// TwinCAT 3 PLC project FRA3
// libraries:
//   Tc2_DataExchange, * (Beckhoff Automation GmbH)
//   Tc2_Standard, * (Beckhoff Automation GmbH)
//   Tc2_System, * (Beckhoff Automation GmbH)
//   Tc2_Utilities, * (Beckhoff Automation GmbH)
//   Tc3_Module, * (Beckhoff Automation GmbH)
//   VisuSymbols,3.5.10.0,System
// project tree:
//   Global Variables/ Global_Variables.TcGVL, Global_Variables_HMI.TcGVL, GVAR_Control.TcGVL, GVAR_Status_and_Alarms.TcGVL, Variable_Configuration.TcGVL
//   POUs/ Control.TcPOU, Hopper_Level.TcPOU, MAIN.TcPOU, Messages.TcPOU, Production_Runtime_Values.TcPOU, Runtime_Control.TcPOU, Speed_Setpoints.TcPOU, StandardCPM.TcPOU, Status_and_Alarms.TcPOU
//   POUs/Function Blocks/ CheckDiv_1.TcPOU, Codes_StopReason.TcPOU, CounterEx.TcPOU, FB_Downtime_LOG.TcPOU, FillerCPM_Current.TcPOU, FixedSchedule_FillerRoom.TcPOU, GetTime_Seconds.TcPOU, LimitRealNumber.TcPOU, LimitRealNumberToWord.TcPOU, ScaleWithParameters.TcPOU, StandardCPMSet.TcPOU, TOGGLE.TcPOU
//   / Standard.TcTTO
// real-time tasks:
//   TASK Standard: cycle T#10ms, priority 20, ADS port 350
// I/O:
//   DEVICE FRA 3 I/O, AmsNetId 5.176.210.24.2.1
//     Term 1 (EK1200) [EK1200-7000 EtherCAT Power supply (1,5A E-Bus)]
//       Term 2 (EL1018) [EL1018 8Ch. Dig. Input 24V, 10µs]
//       Term 3 (EL1018) [EL1018 8Ch. Dig. Input 24V, 10µs]
//       Term 4 (EL1018) [EL1018 8Ch. Dig. Input 24V, 10µs]
//       Term 5 (EL4022) [EL4022 2Ch. Ana. Output 4-20mA, 12bit]
//       Term 6 (EL4022) [EL4022 2Ch. Ana. Output 4-20mA, 12bit]
//       Term 7 (EL4022) [EL4022 2Ch. Ana. Output 4-20mA, 12bit]
//       Term 8 (EL4022) [EL4022 2Ch. Ana. Output 4-20mA, 12bit]
//       Term 9 (EL4022) [EL4022 2Ch. Ana. Output 4-20mA, 12bit]
//       Term 10 (EL4022) [EL4022 2Ch. Ana. Output 4-20mA, 12bit]
//       Term 11 (EL3052) [EL3052 2Ch. Ana. Input 4-20mA]
//       Term 12 (EL3202) [EL3202 2Ch. Ana. Input PT100 (RTD)]
//       Term 13 (EL9110) [EL9110 Power Supplier with LED (24V, Diagnostics)]
//       Term 14 (EL9160) [EL9160 Power Supplier with LED (230V, Diagnostics)]
//       Term 15 (EL2602) [EL2602 2Ch. Relay Output, NO (230V AC / 30V DC)]
//       Term 16 (EL2602) [EL2602 2Ch. Relay Output, NO (230V AC / 30V DC)]
//       Term 17 (EL2602) [EL2602 2Ch. Relay Output, NO (230V AC / 30V DC)]
//       Term 18 (EL2612) [EL2612 2Ch. Relay Output, CO (125V AC / 30V DC)]
//       Term 19 (EL2612) [EL2612 2Ch. Relay Output, CO (125V AC / 30V DC)]
//       Term 20 (EL2612) [EL2612 2Ch. Relay Output, CO (125V AC / 30V DC)]
//       Term 21 (EL2612) [EL2612 2Ch. Relay Output, CO (125V AC / 30V DC)]
//       Term 22 (EL2612) [EL2612 2Ch. Relay Output, CO (125V AC / 30V DC)]
//       Term 23 (EL2612) [EL2612 2Ch. Relay Output, CO (125V AC / 30V DC)]
//       Term 24 (EL2612) [EL2612 2Ch. Relay Output, CO (125V AC / 30V DC)]
//       Term 25 (EL2612) [EL2612 2Ch. Relay Output, CO (125V AC / 30V DC)]
//       Term 26 (EL2612) [EL2612 2Ch. Relay Output, CO (125V AC / 30V DC)]
//       Term 27 (EL9011) [EL9011 End Terminal]
// variable links:
//   FRA3/FRA3 Instance <-> FRA 3 I/O/Term 1 (EK1200)/Term 10 (EL4022)
//     Standard Outputs/.oBrine_Tank_Steam <-> AO Outputs Channel 2/.oBrine_Tank_Steam
//     Standard Outputs/.oSpiral_Infeed_Spd <-> AO Outputs Channel 1/.oSpiral_Infeed_Spd
//   FRA3/FRA3 Instance <-> FRA 3 I/O/Term 1 (EK1200)/Term 11 (EL3052)
//     Standard Inputs/.iHopper_Level <-> AI Standard Channel 1/.iHopper_Level
//   FRA3/FRA3 Instance <-> FRA 3 I/O/Term 1 (EK1200)/Term 12 (EL3202)
//     Standard Inputs/.i1062 <-> RTD Inputs Channel 2/.i1062
//     Standard Inputs/.iSpice_Tank_Temp <-> RTD Inputs Channel 1/.iSpice_Tank_Temp
//   FRA3/FRA3 Instance <-> FRA 3 I/O/Term 1 (EK1200)/Term 14 (EL9160)
//     Standard Inputs/.iEmergency_Stop <-> PowerOK/.iEmergency_Stop
//   FRA3/FRA3 Instance <-> FRA 3 I/O/Term 1 (EK1200)/Term 15 (EL2602)
//     Standard Outputs/.oPreBrine_Flap <-> Channel 2/.oPreBrine_Flap
//     Standard Outputs/.oReturn_Pump <-> Channel 1/.oReturn_Pump
//   FRA3/FRA3 Instance <-> FRA 3 I/O/Term 1 (EK1200)/Term 16 (EL2602)
//     Standard Outputs/.oPre_Brine <-> Channel 1/.oPre_Brine
//     Standard Outputs/.oWater_Valve <-> Channel 2/.oWater_Valve
//   FRA3/FRA3 Instance <-> FRA 3 I/O/Term 1 (EK1200)/Term 17 (EL2602)
//     Standard Outputs/.oBrine_Flap <-> Channel 2/.oBrine_Flap
//     Standard Outputs/.oCloser_Clutch_Sol <-> Channel 1/.oCloser_Clutch_Sol
//   FRA3/FRA3 Instance <-> FRA 3 I/O/Term 1 (EK1200)/Term 18 (EL2612)
//     Standard Outputs/.o1801 <-> Channel 2/.o1801
//     Standard Outputs/.oSpiral_Infeed <-> Channel 1/.oSpiral_Infeed
//   FRA3/FRA3 Instance <-> FRA 3 I/O/Term 1 (EK1200)/Term 19 (EL2612)
//     Standard Outputs/.oCloser <-> Channel 2/.oCloser
//     Standard Outputs/.oSpiral <-> Channel 1/.oSpiral
//   FRA3/FRA3 Instance <-> FRA 3 I/O/Term 1 (EK1200)/Term 2 (EL1018)
//     Standard Inputs/.F_Closer <-> Channel 2/.F_Closer
//     Standard Inputs/.F_Elevator <-> Channel 1/.F_Elevator
//     Standard Inputs/.F_Empty_Can_Conv <-> Channel 8/.F_Empty_Can_Conv
//     Standard Inputs/.F_Empty_Can_Track <-> Channel 7/.F_Empty_Can_Track
//     Standard Inputs/.F_Engler_Filler <-> Channel 5/.F_Engler_Filler
//     Standard Inputs/.F_Full_Can_Belt <-> Channel 3/.F_Full_Can_Belt
//     Standard Inputs/.F_Juicer <-> Channel 4/.F_Juicer
//     Standard Inputs/.F_Twin_Auger <-> Channel 6/.F_Twin_Auger
//   FRA3/FRA3 Instance <-> FRA 3 I/O/Term 1 (EK1200)/Term 20 (EL2612)
//     Standard Outputs/.oFull_Can_Belt <-> Channel 1/.oFull_Can_Belt
//     Standard Outputs/.oJuicer <-> Channel 2/.oJuicer
//   FRA3/FRA3 Instance <-> FRA 3 I/O/Term 1 (EK1200)/Term 21 (EL2612)
//     Standard Outputs/.oEngler_Filler <-> Channel 1/.oEngler_Filler
//     Standard Outputs/.oTwin_Auger_Forward <-> Channel 2/.oTwin_Auger_Forward
//   FRA3/FRA3 Instance <-> FRA 3 I/O/Term 1 (EK1200)/Term 22 (EL2612)
//     Standard Outputs/.oOutfeed_Can_Belt <-> Channel 2/.oOutfeed_Can_Belt
//     Standard Outputs/.oTwin_Auger_Reverse <-> Channel 1/.oTwin_Auger_Reverse
//   FRA3/FRA3 Instance <-> FRA 3 I/O/Term 1 (EK1200)/Term 23 (EL2612)
//     Standard Outputs/.oEmpty_Can_Conv <-> Channel 2/.oEmpty_Can_Conv
//     Standard Outputs/.oEmpty_Can_Track <-> Channel 1/.oEmpty_Can_Track
//   FRA3/FRA3 Instance <-> FRA 3 I/O/Term 1 (EK1200)/Term 24 (EL2612)
//     Standard Outputs/.oInfeed_Auger_Fwd <-> Channel 1/.oInfeed_Auger_Fwd
//     Standard Outputs/.oInfeed_Auger_Rev <-> Channel 2/.oInfeed_Auger_Rev
//   FRA3/FRA3 Instance <-> FRA 3 I/O/Term 1 (EK1200)/Term 25 (EL2612)
//     Standard Outputs/.oCloser_ButtonLt <-> Channel 2/.oCloser_ButtonLt
//     Standard Outputs/.oStatusLt <-> Channel 1/.oStatusLt
//   FRA3/FRA3 Instance <-> FRA 3 I/O/Term 1 (EK1200)/Term 26 (EL2612)
//     Standard Outputs/.oPreBrine_Overflow_Pump <-> Channel 2/.oPreBrine_Overflow_Pump
//     Standard Outputs/.oSpiral_ButtonLt <-> Channel 1/.oSpiral_ButtonLt
//   FRA3/FRA3 Instance <-> FRA 3 I/O/Term 1 (EK1200)/Term 3 (EL1018)
//     Standard Inputs/.F_Exit_Conveyor <-> Channel 6/.F_Exit_Conveyor
//     Standard Inputs/.F_Infeed_Auger <-> Channel 7/.F_Infeed_Auger
//     Standard Inputs/.i403 <-> Channel 8/.i403
//     Standard Inputs/.iCloser_Can_Jam <-> Channel 5/.iCloser_Can_Jam
//     Standard Inputs/.iCloser_Start_PB <-> Channel 2/.iCloser_Start_PB
//     Standard Inputs/.iElevator_Start_PB <-> Channel 3/.iElevator_Start_PB
//     Standard Inputs/.iEmpty_Can_Sensor <-> Channel 4/.iEmpty_Can_Sensor
//     Standard Inputs/.iSpice_Tank_Level <-> Channel 1/.iSpice_Tank_Level
//   FRA3/FRA3 Instance <-> FRA 3 I/O/Term 1 (EK1200)/Term 4 (EL1018)
//     Standard Inputs/.i601 <-> Channel 6/.i601
//     Standard Inputs/.i602 <-> Channel 7/.i602
//     Standard Inputs/.iCloser_Speed_Pulse <-> Channel 8/.iCloser_Speed_Pulse
//     Standard Inputs/.iDischarge_Can_Jam <-> Channel 2/.iDischarge_Can_Jam
//     Standard Inputs/.iElevator_Jam_Sensor <-> Channel 1/.iElevator_Jam_Sensor
//     Standard Inputs/.iPreBrine_Tank_Level <-> Channel 3/.iPreBrine_Tank_Level
//     Standard Inputs/.iSpiral_Can_Counter <-> Channel 5/.iSpiral_Can_Counter
//     Standard Inputs/.iSteamPressSwitch <-> Channel 4/.iSteamPressSwitch
//   FRA3/FRA3 Instance <-> FRA 3 I/O/Term 1 (EK1200)/Term 5 (EL4022)
//     Standard Outputs/.oCloser_Speed <-> AO Outputs Channel 2/.oCloser_Speed
//     Standard Outputs/.oSpice_Pump_Speed <-> AO Outputs Channel 1/.oSpice_Pump_Speed
//   FRA3/FRA3 Instance <-> FRA 3 I/O/Term 1 (EK1200)/Term 6 (EL4022)
//     Standard Outputs/.oElevator_Speed <-> AO Outputs Channel 1/.oElevator_Speed
//     Standard Outputs/.oFull_Can_Belt_Speed <-> AO Outputs Channel 2/.oFull_Can_Belt_Speed
//   FRA3/FRA3 Instance <-> FRA 3 I/O/Term 1 (EK1200)/Term 7 (EL4022)
//     Standard Outputs/.oEngler_Filler_Speed <-> AO Outputs Channel 1/.oEngler_Filler_Speed
//     Standard Outputs/.oTwin_Auger_Speed <-> AO Outputs Channel 2/.oTwin_Auger_Speed
//   FRA3/FRA3 Instance <-> FRA 3 I/O/Term 1 (EK1200)/Term 8 (EL4022)
//     Standard Outputs/.oEmpty_Can_Track_Spd <-> AO Outputs Channel 2/.oEmpty_Can_Track_Spd
//     Standard Outputs/.oExit_Conv_Speed <-> AO Outputs Channel 1/.oExit_Conv_Speed
//   FRA3/FRA3 Instance <-> FRA 3 I/O/Term 1 (EK1200)/Term 9 (EL4022)
//     Standard Outputs/.oEmpty_Can_Conv_Spd <-> AO Outputs Channel 1/.oEmpty_Can_Conv_Spd
//     Standard Outputs/.oInfeed_Auger <-> AO Outputs Channel 2/.oInfeed_Auger

CONFIGURATION FRA3
    RESOURCE PLC ON TwinCAT3
        TASK Standard(INTERVAL := T#10ms, PRIORITY := 20);
        PROGRAM MAIN WITH Standard : MAIN;
    END_RESOURCE
END_CONFIGURATION

// ---- Global Variables/Global_Variables.TcGVL
{attribute 'Tc2GvlVarNames'}
VAR_GLOBAL 
(*****Fill Room A-2****)

(****Slot 1 KL-3052****)
	iHopper_Level AT %I* : WORD;
	i004 AT %I* : WORD;

(****Slot 2 KL-1114****)
	F_Elevator AT %I* : BOOL;
	F_Closer AT %I* : BOOL;
	F_Full_Can_Belt AT %I* : BOOL;
	F_Juicer AT %I* : BOOL;

(****Slot 3 KL-1114****)
	F_Engler_Filler AT %I* : BOOL;
	F_Twin_Auger AT %I* : BOOL;
	F_Empty_Can_Track AT %I* : BOOL;
	F_Empty_Can_Conv AT %I* : BOOL;

(****Slot 4 KL-1114****)
	iSpice_Tank_Level AT %I* : BOOL;
	iCloser_Start_PB AT %I* : BOOL;
	iElevator_Start_PB AT %I* : BOOL;
	iEmpty_Can_Sensor AT %I* : BOOL;

(****Slot 5 KL-1114****)
	iCloser_Can_Jam AT %I* : BOOL;
	F_Exit_Conveyor AT %I* : BOOL;
	F_Infeed_Auger AT %I* : BOOL;
	i403 AT %I* : BOOL;

(****Slot 6 KL-1114****)
	iElevator_Jam_Sensor AT %I* : BOOL;
	iDischarge_Can_Jam AT %I* : BOOL;
	iPreBrine_Tank_Level AT %I* : BOOL;
	iSteamPressSwitch AT %I* : BOOL;

(****Slot 7 KL-1114****)
	iSpiral_Can_Counter AT %I* : BOOL;
	i601 AT %I* : BOOL;
	i602 AT %I* : BOOL;
	iCloser_Speed_Pulse AT %I* : BOOL;

(****Slot 8 KL-4022****)
	oSpice_Pump_Speed AT %Q* : WORD;
	oCloser_Speed AT %Q* : WORD;

(****Slot 9 KL-4022****)
	oElevator_Speed AT %Q* : WORD;
	oFull_Can_Belt_Speed AT %Q* : WORD;

(****Slot 10 KL-4022****)
	oEngler_Filler_Speed AT %Q* : WORD;
	oTwin_Auger_Speed AT %Q* : WORD;

(****Slot 11 KL-4022****)
	oExit_Conv_Speed AT %Q* : WORD;
	oEmpty_Can_Track_Spd AT %Q* : WORD;

(****Slot 12 KL-4022****)
	oEmpty_Can_Conv_Spd AT %Q* : WORD;
	oInfeed_Auger AT %Q* : WORD;

(****Slot 13 KL-4022****)
	oSpiral_Infeed_Spd AT %Q* : WORD;
	oBrine_Tank_Steam AT %Q* : WORD;
	
(****Slot 15 KL-3052****)
	iTwinAugerLVL AT %I* : WORD;
	iSpare AT %I* : WORD;
	
(****Slot 14 KL-3202****)
	iSpice_Tank_Temp AT %I* : WORD;
	i1062 AT %I* : WORD;



(****Slot 16 KL-9260****)
	iEmergency_Stop AT %I* : BOOL;
	iPower AT %I* : BOOL;

(****Slot 17 KL-2602****)
	oReturn_Pump AT %Q* : BOOL;
	oPreBrine_Flap AT %Q* : BOOL;

(****Slot 18 KL-2602****)
	oPre_Brine AT %Q* : BOOL;
	oWater_Valve AT %Q* : BOOL;

(****Slot 19 KL-2602****)
	oCloser_Clutch_Sol AT %Q* : BOOL;
	oBrine_Flap AT %Q* : BOOL;

(****Slot 20 KL-2612****)
	oSpiral_Infeed AT %Q* : BOOL;
	o1801 AT %Q* : BOOL;

(****Slot 21 KL-2612****)
	oSpiral AT %Q* : BOOL;
	oCloser AT %Q* : BOOL;

(****Slot 22 KL-2612****)
	oFull_Can_Belt AT %Q* : BOOL;
	oJuicer AT %Q* : BOOL;

(****Slot 23 KL-2612****)
	oEngler_Filler AT %Q* : BOOL;
	oTwin_Auger_Forward AT %Q* : BOOL;

(****Slot 24 KL-2612****)
	oTwin_Auger_Reverse AT %Q* : BOOL;
	oOutfeed_Can_Belt AT %Q* : BOOL;

(****Slot 25 KL-2612****)
	oEmpty_Can_Track AT %Q* : BOOL;
	oEmpty_Can_Conv AT %Q* : BOOL;

(****Slot 26 KL-2612****)
	oInfeed_Auger_Fwd AT %Q* : BOOL;
	oInfeed_Auger_Rev AT %Q* : BOOL;

(****Slot 27 KL-2612****)
	oStatusLt AT %Q* : BOOL;
	oCloser_ButtonLt AT %Q* : BOOL;

(****Slot 28 KL-2612****)
	oSpiral_ButtonLt AT %Q* : BOOL;
	oPreBrine_Overflow_Pump AT %Q* : BOOL;

	Low_Spice_Alarm: BOOL;
	Low_Spice_Disable: BOOL;
	CleanMode: BOOL;
	Hopper_Level_PCT: REAL;
	TYLER: BOOL;
	Hopper_Level_High: BOOL;
	Brine_Temp_High: BOOL;
	Brine_Temp_Low: BOOL;
	Brine_Temp_Out_Of_Range: BOOL;
	Closer_Steam_Low_Disable: BOOL;
	CanCounter3: CTU;
	CC3Multiplier: CTU;
	DowntimeTotal_Min: REAL;
	EndRuntime: BOOL;
	AutoTog: TOGGLE;
	FillerPauseTog: TOGGLE;
	FillerAugerPause: TOGGLE;
	Empty_Can_Tog: TOGGLE;
	CC3Reset: BOOL;
	CanCntReset: BOOL;
	Count3: WORD;
    Runtime_Stopped: BOOL;
	Count3Real: REAL;
	MultiReal: REAL;
	HighCount: REAL;
	ActualCount: REAL;
	Cases: REAL;
    MultiWord: WORD ;

END_VAR

// ---- Global Variables/Global_Variables_HMI.TcGVL
{attribute 'Tc2GvlVarNames'}
VAR_GLOBAL

	s3ProdStd:REAL;

(*Speed Set Points*)
	sSpice_Pump_Speed_SPt: REAL;
	sCloser_Speed_SPt: REAL;
	sElevator_Speed_SPt: REAL;
	sFull_Can_Belt_Speed_SPt: REAL;
	sEngler_Filler_Speed_SPt: REAL;
	sTwin_Auger_Speed_SPt: REAL;
	sExit_Conveyor_Speed_SPt: REAL;
	Empty_Can_Track_SPt: REAL;
	Empty_Can_Conv_SPt: REAL;
	sInfeed_Auger_SPt: REAL;

(****Screen Activation****)

	sAuto: BOOL;
	sAuto_Run:BOOL;
	sAuto_Button : BOOL;
	sFiller_Pause_Button : BOOL;
	sFiller_Pause : BOOL;
	sFeed_Auger_Pause_Button : BOOL;
	sFeed_Auger_Pause : BOOL;
	sEmpty_Can_Track : BOOL;

	sFeed_Auger_Fwd : BOOL;
	sFeed_Auger_Rev : BOOL;
	sTwin_Auger_Fwd : BOOL;
	sTwin_Auger_Rev : BOOL;

	oInfeed_Auger_Fwd_Light: BOOL;
	oInfeed_Auger_Rev_Light: BOOL;
	oTwin_Auger_Forward_Light: BOOL;
	oTwin_Auger_Reverse_Light: BOOL;
	Jam_Fault: BOOL;
	sEngler_Filler : BOOL;
	sPreBrine : BOOL;
	sSpice_Tank_Fill : BOOL;
	sConveyors : BOOL;
	sJuicer : BOOL;
	sDiverter : BOOL;
	sEmpty_Can_Track_300A: BOOL;
	sCloser: BOOL;
	sFull_Can_Belt: BOOL;
	sPre_Brine: BOOL;
	sSpice_Diverter: BOOL;
	sCloser_Current: REAL;
	sEmpty_Can_Conv: BOOL;
	Auto_Run: BOOL;



	sMessages: STRING;
	Spice_Tank_Temp_F: REAL;
	sEmpty_Can_Track_Light : BOOL;

	sManualFillJuicerButton: BOOL;
	sManualFillJuicerButton_Light: BOOL;

	sSteam_Enable: BOOL;
	sSteam_Enable_Lt: BOOL;

	sSpice_Temp_SetPoint: REAL;
	sBrineTempF: REAL;
	sBrine_Tank_Steam: REAL;

	sWater_Valve_enable : BOOL;
	sSpice_Valve_enable : BOOL;
	sSpice_Valve_enable_Lt: BOOL;
	sWater_Valve_enable_Lt: BOOL;

	sCleanMode: BOOL;
	sCleanMode_Light: BOOL;

	sCloser_Steam_ON: BOOL;
	sCloserSteamEnable: BOOL;
	sCloserSteamEnable_Lt: BOOL;


(**HMI Access Code Variables**)

	sButton1:INT:=7390;
	sButton2:INT:=23520;
	sButton3:INT:=1258;
	sButton4:INT:=1225;
	sButton5:INT:=7680;
	sButton6:INT:=12281;
	sButton7:INT:=5746;
	sButton8:INT:=15051;
	sButton9:INT:=3341;
	sButton10:INT:=12159;
	sButton11:INT:=12310;
	sButton12:INT:=11490;
	sButton13:INT:=1522;
	sButton14:INT:=0596;
	sButton15:INT:=22548;
	sButton16:INT:=15293;
	sButton17:INT:=15108;
	sButton18:INT:=430;
	sButton19:INT:=2668;
	sButton20:INT:=12396;
	sButton21:INT:=7171;
	sButton22:INT:=7272;
	sButton23:INT:=7373;
	sButton24:INT:=7474;

(**************Scada Comms*********************)
	sc3_Current_CPM:INT;
	sc3_CPM_AVG:REAL;
	sc3ActualCount: REAL;
	sc3_BackupCouter_ActualCount: DINT;
	sc3_Opt:REAL;
	sc3_EFF: REAL;
    CounterEx_0: CounterEx;
    CounterEx_1: CounterEx;
	CounterEx_2: CounterEx;

    sc3CloserSpeedCPM: INT;

	sc3_Running: BOOL;
	sc3_Spiral_Drive_Fault: BOOL;
	sc3_Elevator_Drive_Fault: BOOL;
	sc3_Filler_Drive_Fault: BOOL;
	sc3_Closer8Drive_Fault: BOOL;
	sc3_Hopper_Lvl: BOOL;
	sc3_Alarm_Reset: BOOL;
	sc3_Auger_Fault: BOOL;
	sc3_Spiral_Infeed_Fault: BOOL;
	sc3_Closer_Outfeed_Fault: BOOL;
	sc3_Spiral_Infeed_Belt_Fault: BOOL;
	sc3_Filler_Line_Conv_Fault: BOOL;
	sc3_Brine_Temp_Fault:BOOL;

	sc3_SteamPsi_OK: BOOL;
	sc3_AirPsi_Ok: BOOL;
	sc3_ProdCode:STRING:='2GEBEBB - 300 Bright Peas';


	RPT: REAL;
	Needed_CPM: REAL;
	sc3_CanReset: BOOL;
	rsPlant_Air_Psi: DINT;
	sc3Plant_Air_Psi: DINT;
	rMeasuredSteamPsi: INT;
	sc3Closer_Speed: INT;

	Hopper_Level_Low: BOOL;

	sc3_IgnitionStartProdTime: BOOL;


	FRA3_Hopper_Level: REAL;
	HopperLevel_IS_HIGH: BOOL;
	HopperLevelIS_LOW: BOOL;
	
	(*L3: Downtime Log*)
	sc3_FillerStops: INT;
	sc3_StartProd_Button: BOOL;
	sc3_EndProd_Button: BOOL;
	sc3_ID_Downtime: INT;
	sc3_ConfmirDT_Button: BOOL;
	sc3_Code_DowntimeLog: STRING;
	sc3_DowntimeLog: BOOL;
	sc3_InProduction_Status: BOOL;
	sc3_DowntimeView_Control: BOOL;
	
	(*L3: Uptime & Downtime*)
	sc3_Downtime_SEC: DINT;
	sc3_Uptime_SEC: DINT;
END_VAR

// ---- Global Variables/GVAR_Control.TcGVL
{attribute 'Tc2GvlVarNames'}
VAR_GLOBAL
	CloserTOG: TOGGLE;
	ElevatorTOG: TOGGLE;
	FFAugerTOG: TOGGLE;
	CanBeltTOG: TOGGLE;


	Twin_AugerTOG: TOGGLE;
	Pre_BrineTOG: TOGGLE;
	Diverter_Tog: TOGGLE;
	JuicerTOG: TOGGLE;
	EmptyCanTrackTOG: TOGGLE;
	EnglerFillerTOG: TOGGLE;
	EmptyCanTOG: TOGGLE;
	Fill_Pulse: TP;
	Spice_Tank_ValveTOG: TOGGLE;
	Spice_Tank_Valve_Light: BOOL;
	Auger_Fwd_Momentum_Safety: TOF;
	FFAugerRevTOG: TOGGLE;
	Auger_Rev_Momentum_Safety: TOF;
	Twin_AugerRevTOG: TOGGLE;
	TwinAuger_Fwd_Momentum_Safety: TOF;
	TwinAuger_Rev_Momentum_Safety: TOF;

	Full_CanBelt_Delay: TON;
	CloserJamTMR: TON;
	Jam_Alarm_Maintain: TOF;

	CloserJam2TMR: TON;
	PreBrine_Maintain: TOF;
	CloserJam3TMR: TON;
	Brine_PID: FB_BasicPID;
	Reset_Spice_PID: BOOL;
	Steam_Enable_TOG: TOGGLE;
	Low_Lvl_Juicer_Alarm_TMR: TON;
	Solbern_Maintain_During_Low_Spice: TON;
	RefillJuicer: TOGGLE;
	JuicerLowLevelDelay: TON;
	No_Cans_Delay: TON;
	No_Empty_Cans_Pause: BOOL;
	Water_Valve_Enable_Tog: TOGGLE;
	Spice_Valve_Enable_Tog: TOGGLE;
	CleanModeTOG: TOGGLE;
	Hopper_PID: FB_BasicPID;
	Reset_Hopper_PID: BOOL;
	Hopper_Level_SP: REAL;
	Infeed_Auger_Speed: REAL;
	High_Level_Delay_TMR: TON;
	Infeed_Slow_Delay: TON;
	Infeed_Resume_Delay: TON;
	Brine_Temp_OOR_TMR: TON;
	Water_Delay_OFF: TOF;
	Spice_Delay_OFF: TOF;
	Closer_Steam_Low_Disable_Delay: TON;
	CloserSteamControl_Tog: TOGGLE;
	Hopper_High_Delay: TON;
	Hopper_High_Mtain: TOF;
	HHM: TIME;
	Infeed_Low_Speed: BOOL;

	Hopper_Low_LevelTMR: TON;
	HopperLow_TT: TIME;
	Hop_Low_Lvl_DebounceTMR: TOF;
	Filler3_Sys_Running: BOOL;
	StopTwinAuger: BOOL;
	AugerStopTMR: TON;
END_VAR

// ---- Global Variables/GVAR_Status_and_Alarms.TcGVL
{attribute 'Tc2GvlVarNames'}
VAR_GLOBAL
END_VAR

// ---- Global Variables/Variable_Configuration.TcGVL
{attribute 'Tc2GvlVarNames'}
VAR_CONFIG
END_VAR

// ---- POUs/MAIN.TcPOU
PROGRAM MAIN
VAR

	
	FCV_1: INT;
	FCV_2: INT;
	HopperLevel: REAL;
END_VAR

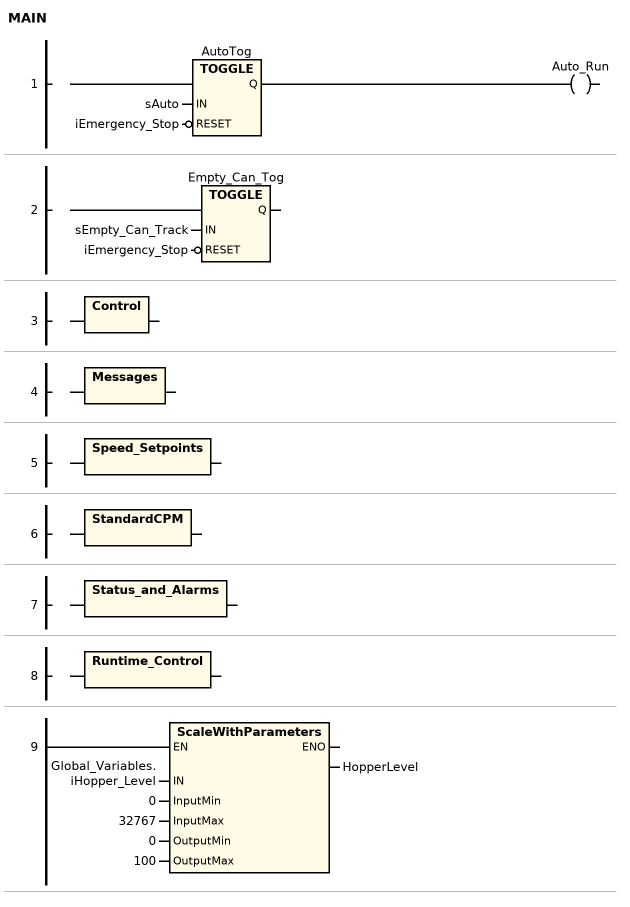
// NETWORK 1
AutoTog(IN := sAuto, RESET := NOT iEmergency_Stop); // TOGGLE
Auto_Run := AutoTog.Q;

// NETWORK 2
Empty_Can_Tog(IN := sEmpty_Can_Track, RESET := NOT iEmergency_Stop); // TOGGLE

// NETWORK 3
Control();

// NETWORK 4
Messages();

// NETWORK 5
Speed_Setpoints();

// NETWORK 6
StandardCPM();

// NETWORK 7
Status_and_Alarms();

// NETWORK 8
Runtime_Control();

// NETWORK 9
HopperLevel := ScaleWithParameters(IN := Global_Variables.iHopper_Level, InputMin := 0, InputMax := 32767, OutputMin := 0, OutputMax := 100);

END_PROGRAM

// ---- POUs/Function Blocks/TOGGLE.TcPOU
FUNCTION_BLOCK TOGGLE
VAR_INPUT
	IN : BOOL;
	RESET : BOOL;
END_VAR
VAR_OUTPUT
	Q : BOOL;
END_VAR
VAR
	edge : BOOL;
END_VAR

(* This function block toggle the state of the output (Q) when the input (IN)
	transitions from a FALSE to TRUE.
	If the reset input (RESET) is true, then the output is always false *)
IF RESET THEN
	Q:=0;
ELSIF IN AND NOT edge THEN
	Q:=NOT Q;
END_IF;
edge:=IN;

END_FUNCTION_BLOCK

// ---- POUs/Control.TcPOU
PROGRAM Control
VAR


	ToggleSpiral: TOGGLE;
	HopperLevel_High: TON;
	HopperLevelHigh: BOOL;
	HopperLevelLow: BOOL;
	HopperLevelISLow: BOOL;
	HopperLevelISHigh: BOOL;
	Hopper_Level: Hopper_Level;
	Hopper_LevelLow: TON;
	Twin_Auger_Level: Hopper_Level;
	FRA3_HopperLevel_INT: INT;
	sSpice_Tank_Valve: BOOL;
	PreBrine_Delay: TON;
	PreBrineValveTON: TON;
	PreBrineValveTOF: TOF;
	Feed: ton;
	Auger: ton;
	FeedAugerResume: ton;
	Resume: BOOL;
	Auger_Resume: BOOL;
	HopperResume: tof;
	FillerCPM: FillerCPM_Current;
	sFillerCPM_Current: REAL;
	HopperLevelLow_Timer: TIME;
	SpareTON_1: TON;
END_VAR
VAR PERSISTENT
	SpareTONTest: BOOL;
	SpareTimerTest: BOOL;
	HopperLevelLowHMI: INT;
	HopperLevelLowCalc: INT;
	HopperLevelHighHMI: INT;
	HopperLevelHighCalc: INT;
	HopperLevelHigh_Timer: TIME;
	FeedAugerResumeHMI: INT;
	FeedAugerResumeCalc: INT;
	FeedAugerDelayHMITimer: TIME;
	sCloserJam_1_RealValue: REAL;
	sCloserJam_1RV: REAL;
	sCloserJam_1PT: TIME;
	sCloserJam_2_RealValue: REAL;
	sCloserJam_2RV: REAL;
	sCloserJam_2PT: TIME;
	sElevatorJam_RealValue: REAL;
	sElevatorJamRV: REAL;
	sElevatorJamPT: TIME;
	sFullCanBeltDelay_RealValue: REAL;
	sFullCanBeltDelayRV: REAL;
	sFullCanBeltDelayPT: TIME;
	sNoEmptyCansDelay_RealValue: REAL;
	sNoEmptyCansDelayRV: REAL;
	sNoEmptyCansDelayPT: TIME;
	sPrebrineFlapON_RealValue: REAL;
	sPrebrineFlapOFFRV: REAL;
	sPrebrineFlapONRV: REAL;
	sPrebrineFlapONPT: TIME;
	sPrebrineFlapOFF_RealValue: REAL;
	sPrebrineFlapOFFPT: TIME;
	sPrebrineValveON_RealValue: REAL;
	sPrebrineValveONRV: REAL;
	sPrebrineValveONPT: TIME;
	sPrebrineValveOFF_RealValue: REAL;
	sPrebrineValveOffRV: REAL;
	sPrebrineValveOffPT: TIME;
	sRefillJuicer_RealValue: REAL;
	sRefillJuicerRV: REAL;
	sRefillJuicerPT: TIME;
	sLowSpiceDisable_RealValue: REAL;
	sLowSpiceDisableRV: REAL;
	sLowSpiceDisablePT: TIME;
END_VAR
VAR // added by the converter: edge detectors and wires of the graphical bodies
    _w1, _w2, _w3 : BOOL;
END_VAR

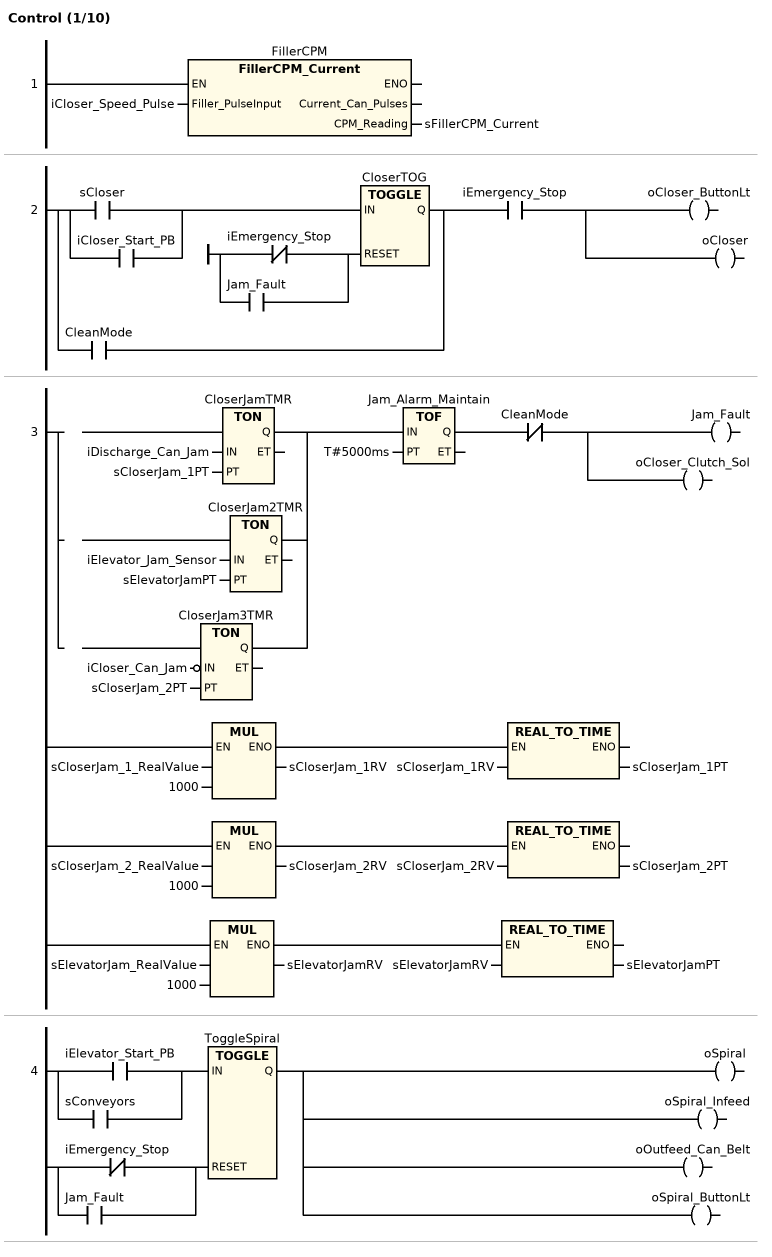
// NETWORK 1
FillerCPM(Filler_PulseInput := iCloser_Speed_Pulse, CPM_Reading => sFillerCPM_Current); // FillerCPM_Current

// NETWORK 2
CloserTOG(IN := sCloser OR iCloser_Start_PB, RESET := NOT iEmergency_Stop OR Jam_Fault); // TOGGLE
_w1 := (CloserTOG.Q OR CleanMode) AND iEmergency_Stop;
oCloser_ButtonLt := _w1;
oCloser := _w1;

// NETWORK 3
CloserJamTMR(IN := iDischarge_Can_Jam, PT := sCloserJam_1PT); // TON
CloserJam2TMR(IN := iElevator_Jam_Sensor, PT := sElevatorJamPT); // TON
CloserJam3TMR(IN := NOT iCloser_Can_Jam, PT := sCloserJam_2PT); // TON
Jam_Alarm_Maintain(IN := CloserJamTMR.Q OR CloserJam2TMR.Q OR CloserJam3TMR.Q, PT := T#5000ms); // TOF
_w2 := Jam_Alarm_Maintain.Q AND NOT CleanMode;
Jam_Fault := _w2;
oCloser_Clutch_Sol := _w2;
sCloserJam_1RV := sCloserJam_1_RealValue * 1000;
sCloserJam_1PT := REAL_TO_TIME(sCloserJam_1RV);
sCloserJam_2RV := sCloserJam_2_RealValue * 1000;
sCloserJam_2PT := REAL_TO_TIME(sCloserJam_2RV);
sElevatorJamRV := sElevatorJam_RealValue * 1000;
sElevatorJamPT := REAL_TO_TIME(sElevatorJamRV);

// NETWORK 4
ToggleSpiral(IN := iElevator_Start_PB OR sConveyors, RESET := NOT iEmergency_Stop OR Jam_Fault); // TOGGLE
oSpiral := ToggleSpiral.Q;
oSpiral_Infeed := ToggleSpiral.Q;
oOutfeed_Can_Belt := ToggleSpiral.Q;
oSpiral_ButtonLt := ToggleSpiral.Q;

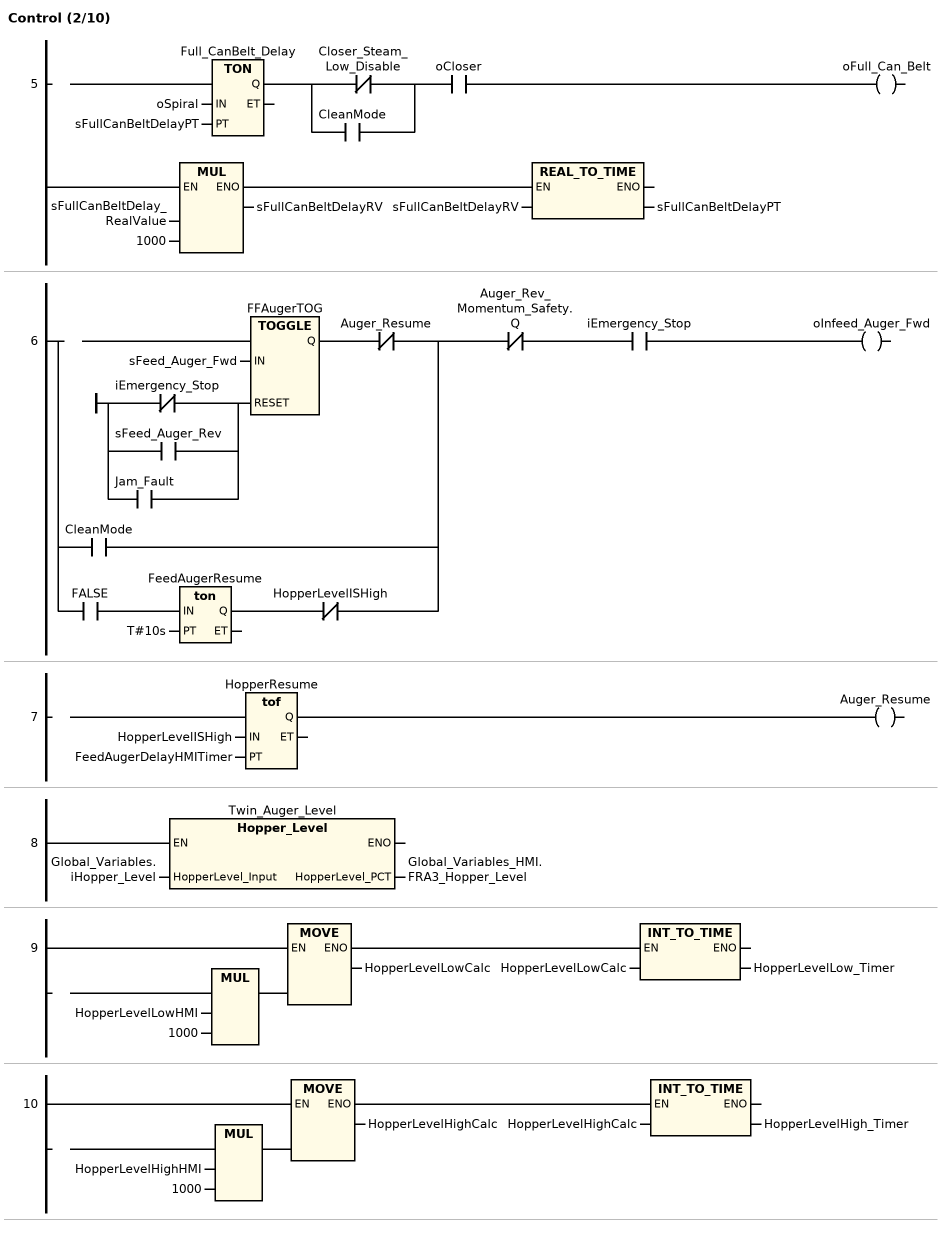
// NETWORK 5
Full_CanBelt_Delay(IN := oSpiral, PT := sFullCanBeltDelayPT); // TON
oFull_Can_Belt := Full_CanBelt_Delay.Q AND (NOT Closer_Steam_Low_Disable OR CleanMode) AND oCloser;
sFullCanBeltDelayRV := sFullCanBeltDelay_RealValue * 1000;
sFullCanBeltDelayPT := REAL_TO_TIME(sFullCanBeltDelayRV);

// NETWORK 6
FFAugerTOG(IN := sFeed_Auger_Fwd, RESET := NOT iEmergency_Stop OR sFeed_Auger_Rev OR Jam_Fault); // TOGGLE
FeedAugerResume(IN := FALSE, PT := T#10s); // ton
oInfeed_Auger_Fwd := (FFAugerTOG.Q AND NOT Auger_Resume OR CleanMode OR FeedAugerResume.Q AND NOT HopperLevelISHigh) AND NOT Auger_Rev_Momentum_Safety.Q AND iEmergency_Stop;

// NETWORK 7
HopperResume(IN := HopperLevelISHigh, PT := FeedAugerDelayHMITimer); // tof
Auger_Resume := HopperResume.Q;

// NETWORK 8
Twin_Auger_Level(HopperLevel_Input := Global_Variables.iHopper_Level, HopperLevel_PCT => Global_Variables_HMI.FRA3_Hopper_Level); // Hopper_Level

// NETWORK 9
HopperLevelLowCalc := HopperLevelLowHMI * 1000;
HopperLevelLow_Timer := INT_TO_TIME(HopperLevelLowCalc);

// NETWORK 10
HopperLevelHighCalc := HopperLevelHighHMI * 1000;
HopperLevelHigh_Timer := INT_TO_TIME(HopperLevelHighCalc);

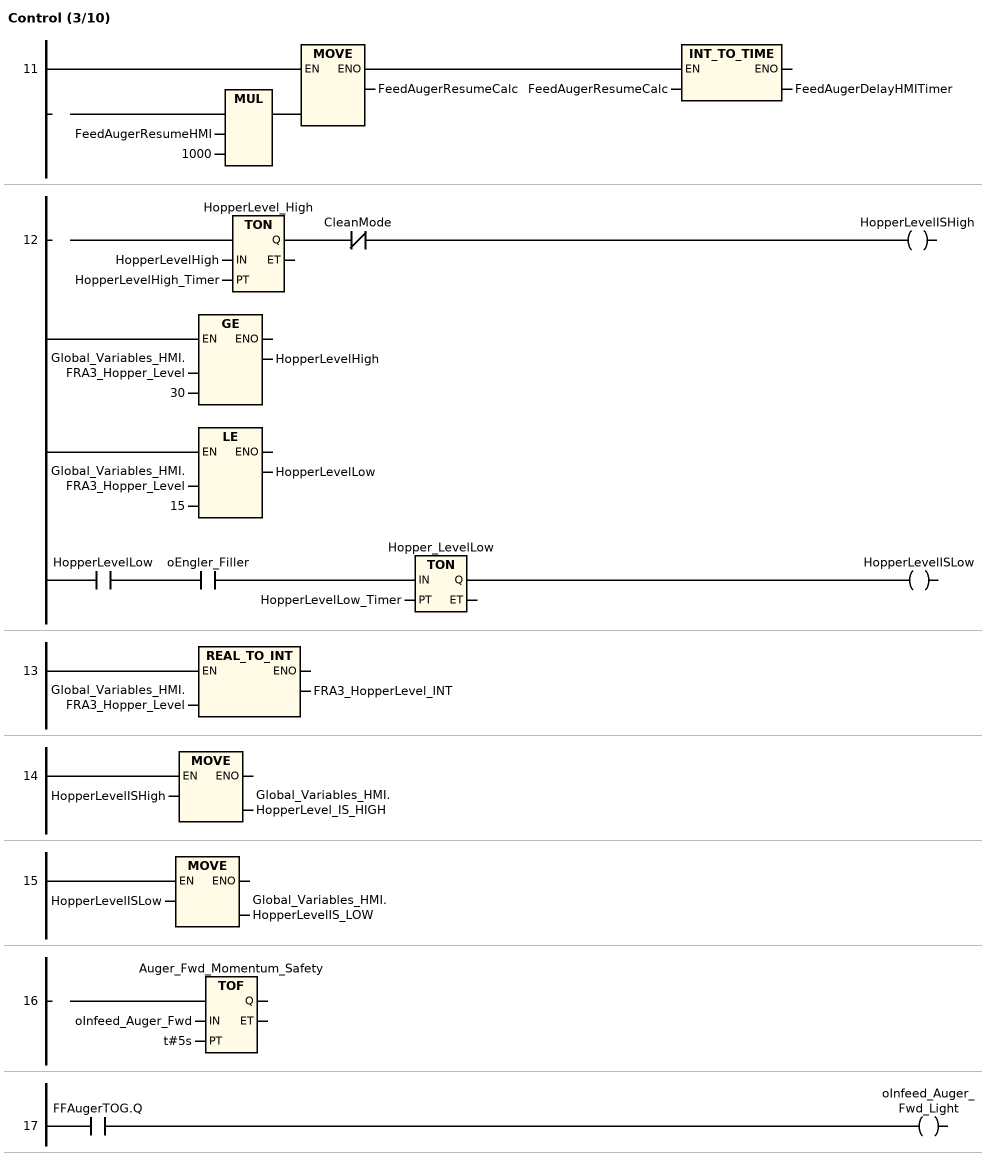
// NETWORK 11
FeedAugerResumeCalc := FeedAugerResumeHMI * 1000;
FeedAugerDelayHMITimer := INT_TO_TIME(FeedAugerResumeCalc);

// NETWORK 12
HopperLevel_High(IN := HopperLevelHigh, PT := HopperLevelHigh_Timer); // TON
HopperLevelISHigh := HopperLevel_High.Q AND NOT CleanMode;
HopperLevelHigh := Global_Variables_HMI.FRA3_Hopper_Level >= 30;
HopperLevelLow := Global_Variables_HMI.FRA3_Hopper_Level <= 15;
Hopper_LevelLow(IN := HopperLevelLow AND oEngler_Filler, PT := HopperLevelLow_Timer); // TON
HopperLevelISLow := Hopper_LevelLow.Q;

// NETWORK 13
FRA3_HopperLevel_INT := REAL_TO_INT(Global_Variables_HMI.FRA3_Hopper_Level);

// NETWORK 14
Global_Variables_HMI.HopperLevel_IS_HIGH := HopperLevelISHigh;

// NETWORK 15
Global_Variables_HMI.HopperLevelIS_LOW := HopperLevelISLow;

// NETWORK 16
Auger_Fwd_Momentum_Safety(IN := oInfeed_Auger_Fwd, PT := t#5s); // TOF

// NETWORK 17
oInfeed_Auger_Fwd_Light := FFAugerTOG.Q;

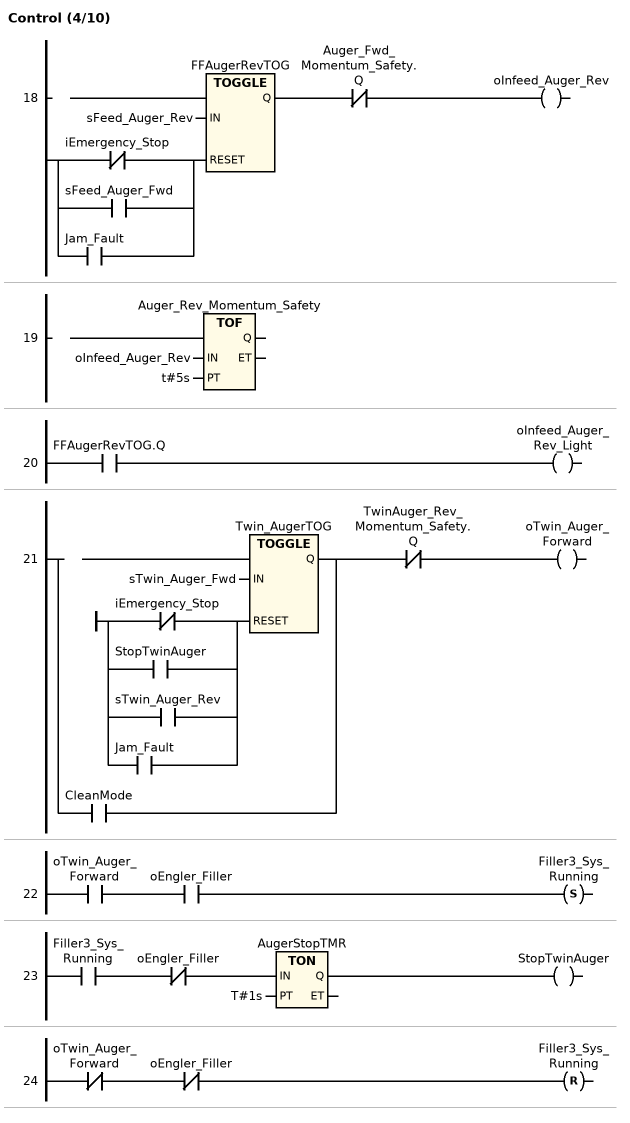
// NETWORK 18
FFAugerRevTOG(IN := sFeed_Auger_Rev, RESET := NOT iEmergency_Stop OR sFeed_Auger_Fwd OR Jam_Fault); // TOGGLE
oInfeed_Auger_Rev := FFAugerRevTOG.Q AND NOT Auger_Fwd_Momentum_Safety.Q;

// NETWORK 19
Auger_Rev_Momentum_Safety(IN := oInfeed_Auger_Rev, PT := t#5s); // TOF

// NETWORK 20
oInfeed_Auger_Rev_Light := FFAugerRevTOG.Q;

// NETWORK 21
Twin_AugerTOG(IN := sTwin_Auger_Fwd, RESET := NOT iEmergency_Stop OR StopTwinAuger OR sTwin_Auger_Rev OR Jam_Fault); // TOGGLE
oTwin_Auger_Forward := (Twin_AugerTOG.Q OR CleanMode) AND NOT TwinAuger_Rev_Momentum_Safety.Q;

// NETWORK 22
Filler3_Sys_Running S= oTwin_Auger_Forward AND oEngler_Filler;

// NETWORK 23
AugerStopTMR(IN := Filler3_Sys_Running AND NOT oEngler_Filler, PT := T#1s); // TON
StopTwinAuger := AugerStopTMR.Q;

// NETWORK 24
Filler3_Sys_Running R= NOT oTwin_Auger_Forward AND NOT oEngler_Filler;

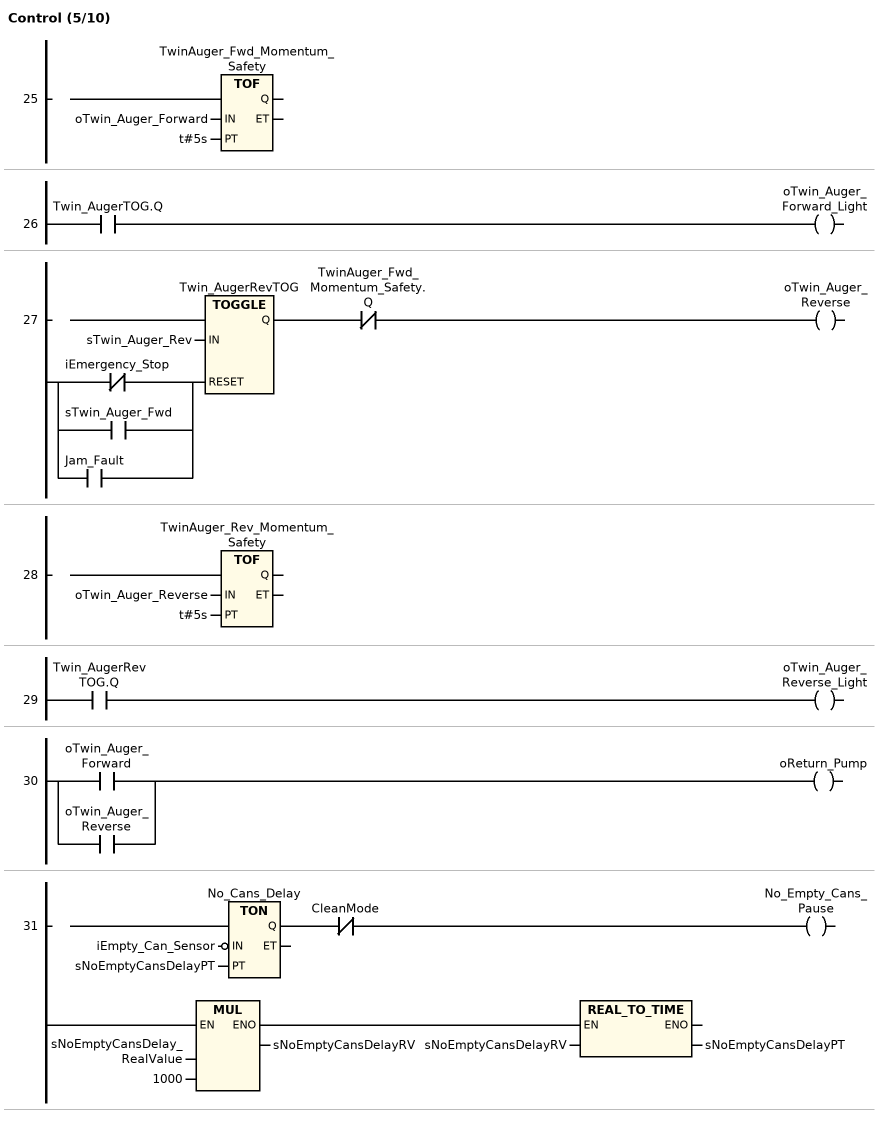
// NETWORK 25
TwinAuger_Fwd_Momentum_Safety(IN := oTwin_Auger_Forward, PT := t#5s); // TOF

// NETWORK 26
oTwin_Auger_Forward_Light := Twin_AugerTOG.Q;

// NETWORK 27
Twin_AugerRevTOG(IN := sTwin_Auger_Rev, RESET := NOT iEmergency_Stop OR sTwin_Auger_Fwd OR Jam_Fault); // TOGGLE
oTwin_Auger_Reverse := Twin_AugerRevTOG.Q AND NOT TwinAuger_Fwd_Momentum_Safety.Q;

// NETWORK 28
TwinAuger_Rev_Momentum_Safety(IN := oTwin_Auger_Reverse, PT := t#5s); // TOF

// NETWORK 29
oTwin_Auger_Reverse_Light := Twin_AugerRevTOG.Q;

// NETWORK 30
oReturn_Pump := oTwin_Auger_Forward OR oTwin_Auger_Reverse;

// NETWORK 31
No_Cans_Delay(IN := NOT iEmpty_Can_Sensor, PT := sNoEmptyCansDelayPT); // TON
No_Empty_Cans_Pause := No_Cans_Delay.Q AND NOT CleanMode;
sNoEmptyCansDelayRV := sNoEmptyCansDelay_RealValue * 1000;
sNoEmptyCansDelayPT := REAL_TO_TIME(sNoEmptyCansDelayRV);

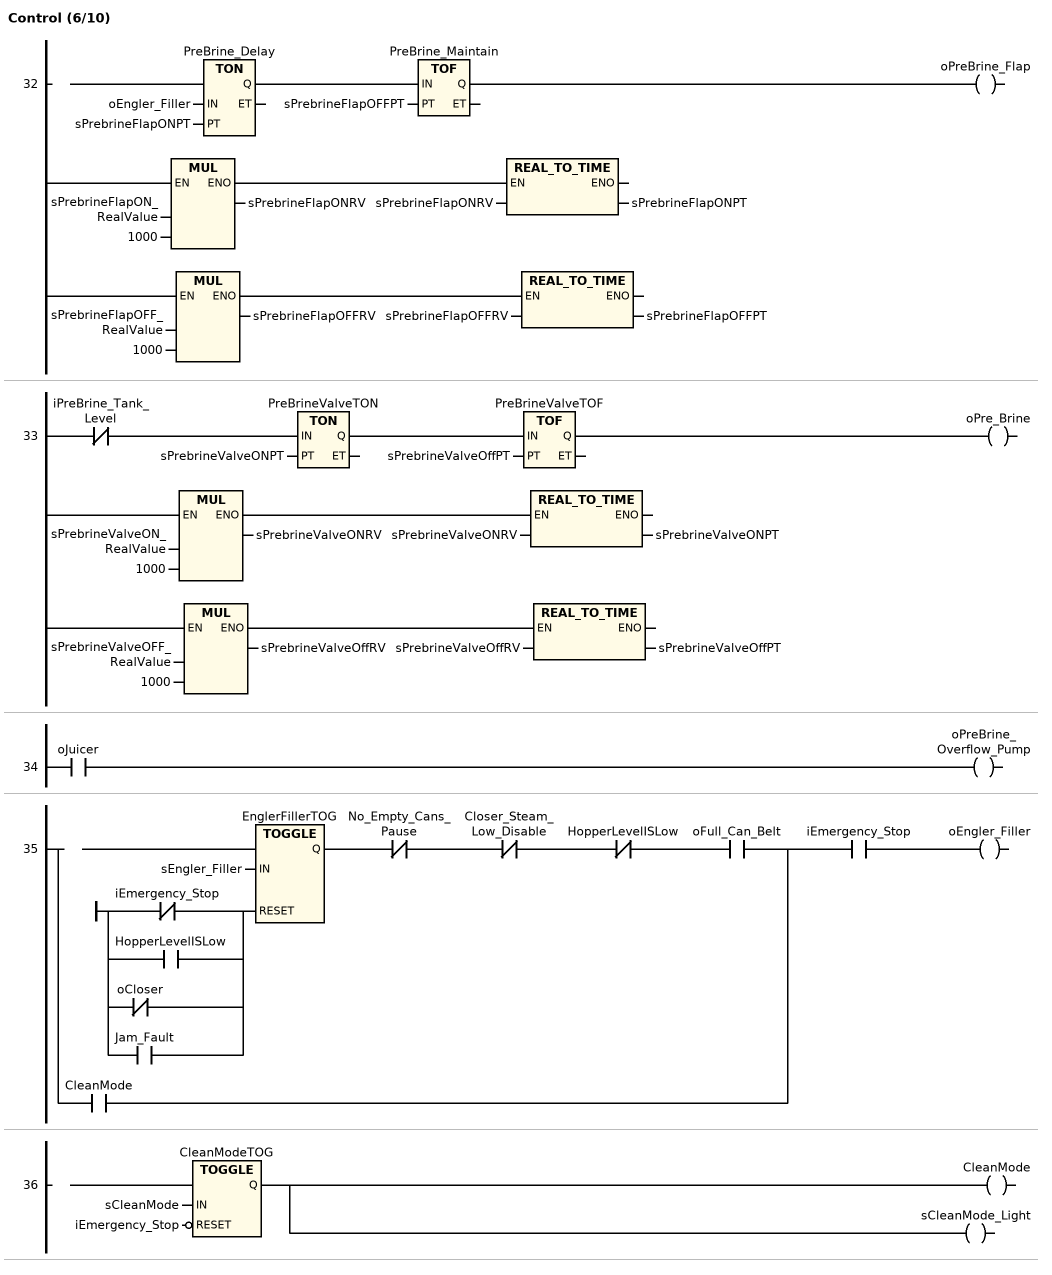
// NETWORK 32
PreBrine_Delay(IN := oEngler_Filler, PT := sPrebrineFlapONPT); // TON
PreBrine_Maintain(IN := PreBrine_Delay.Q, PT := sPrebrineFlapOFFPT); // TOF
oPreBrine_Flap := PreBrine_Maintain.Q;
sPrebrineFlapONRV := sPrebrineFlapON_RealValue * 1000;
sPrebrineFlapONPT := REAL_TO_TIME(sPrebrineFlapONRV);
sPrebrineFlapOFFRV := sPrebrineFlapOFF_RealValue * 1000;
sPrebrineFlapOFFPT := REAL_TO_TIME(sPrebrineFlapOFFRV);

// NETWORK 33
PreBrineValveTON(IN := NOT iPreBrine_Tank_Level, PT := sPrebrineValveONPT); // TON
PreBrineValveTOF(IN := PreBrineValveTON.Q, PT := sPrebrineValveOffPT); // TOF
oPre_Brine := PreBrineValveTOF.Q;
sPrebrineValveONRV := sPrebrineValveON_RealValue * 1000;
sPrebrineValveONPT := REAL_TO_TIME(sPrebrineValveONRV);
sPrebrineValveOffRV := sPrebrineValveOFF_RealValue * 1000;
sPrebrineValveOffPT := REAL_TO_TIME(sPrebrineValveOffRV);

// NETWORK 34
oPreBrine_Overflow_Pump := oJuicer;

// NETWORK 35
EnglerFillerTOG(IN := sEngler_Filler, RESET := NOT iEmergency_Stop OR HopperLevelISLow OR NOT oCloser OR Jam_Fault); // TOGGLE
oEngler_Filler := (EnglerFillerTOG.Q AND NOT No_Empty_Cans_Pause AND NOT Closer_Steam_Low_Disable AND NOT HopperLevelISLow AND oFull_Can_Belt OR CleanMode) AND iEmergency_Stop;

// NETWORK 36
CleanModeTOG(IN := sCleanMode, RESET := NOT iEmergency_Stop); // TOGGLE
CleanMode := CleanModeTOG.Q;
sCleanMode_Light := CleanModeTOG.Q;

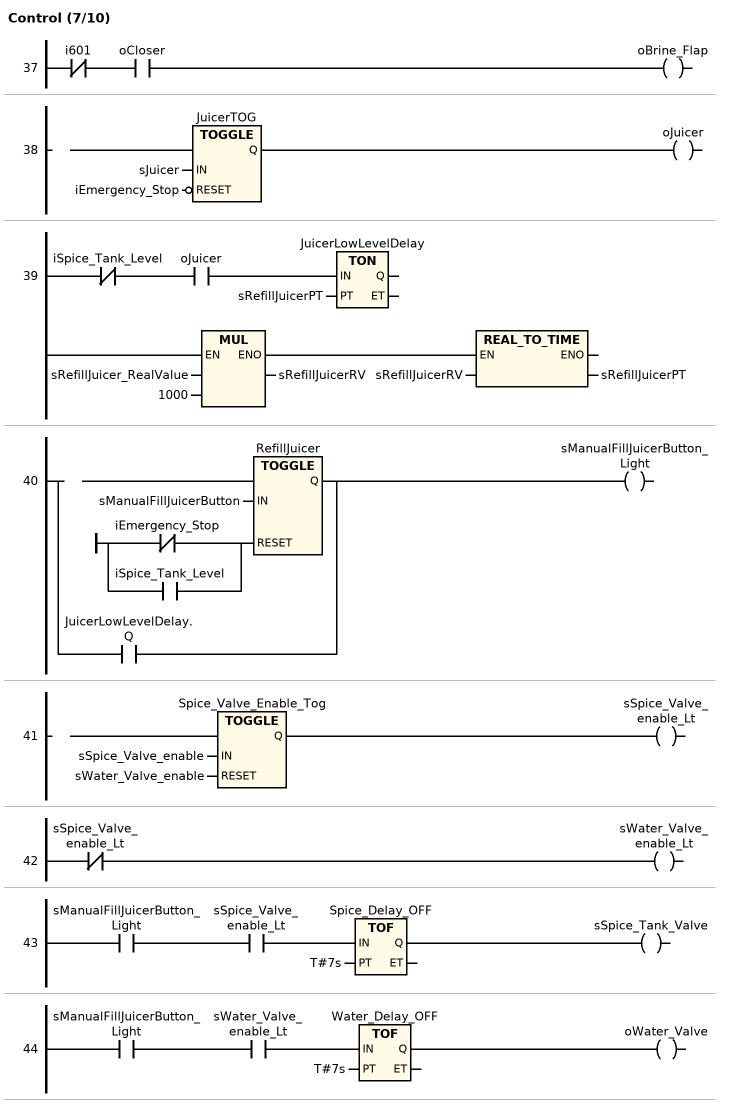
// NETWORK 37
oBrine_Flap := NOT i601 AND oCloser;

// NETWORK 38
JuicerTOG(IN := sJuicer, RESET := NOT iEmergency_Stop); // TOGGLE
oJuicer := JuicerTOG.Q;

// NETWORK 39
JuicerLowLevelDelay(IN := NOT iSpice_Tank_Level AND oJuicer, PT := sRefillJuicerPT); // TON
sRefillJuicerRV := sRefillJuicer_RealValue * 1000;
sRefillJuicerPT := REAL_TO_TIME(sRefillJuicerRV);

// NETWORK 40
RefillJuicer(IN := sManualFillJuicerButton, RESET := NOT iEmergency_Stop OR iSpice_Tank_Level); // TOGGLE
sManualFillJuicerButton_Light := RefillJuicer.Q OR JuicerLowLevelDelay.Q;

// NETWORK 41
Spice_Valve_Enable_Tog(IN := sSpice_Valve_enable, RESET := sWater_Valve_enable); // TOGGLE
sSpice_Valve_enable_Lt := Spice_Valve_Enable_Tog.Q;

// NETWORK 42
sWater_Valve_enable_Lt := NOT sSpice_Valve_enable_Lt;

// NETWORK 43
Spice_Delay_OFF(IN := sManualFillJuicerButton_Light AND sSpice_Valve_enable_Lt, PT := T#7s); // TOF
sSpice_Tank_Valve := Spice_Delay_OFF.Q;

// NETWORK 44
Water_Delay_OFF(IN := sManualFillJuicerButton_Light AND sWater_Valve_enable_Lt, PT := T#7s); // TOF
oWater_Valve := Water_Delay_OFF.Q;

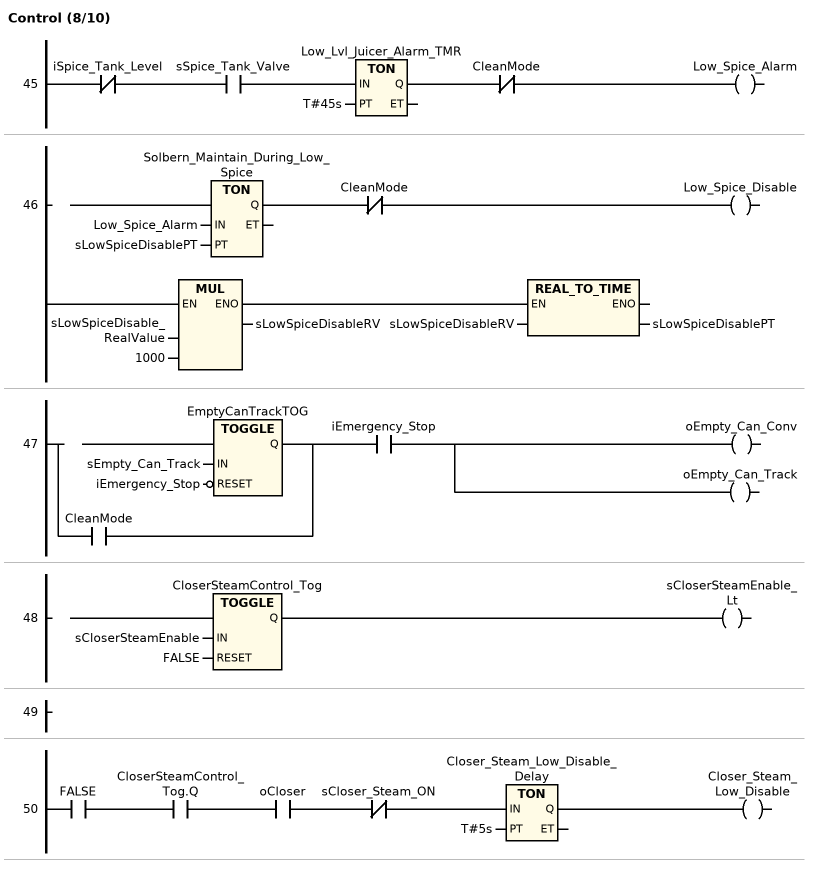
// NETWORK 45
Low_Lvl_Juicer_Alarm_TMR(IN := NOT iSpice_Tank_Level AND sSpice_Tank_Valve, PT := T#45s); // TON
Low_Spice_Alarm := Low_Lvl_Juicer_Alarm_TMR.Q AND NOT CleanMode;

// NETWORK 46
Solbern_Maintain_During_Low_Spice(IN := Low_Spice_Alarm, PT := sLowSpiceDisablePT); // TON
Low_Spice_Disable := Solbern_Maintain_During_Low_Spice.Q AND NOT CleanMode;
sLowSpiceDisableRV := sLowSpiceDisable_RealValue * 1000;
sLowSpiceDisablePT := REAL_TO_TIME(sLowSpiceDisableRV);

// NETWORK 47
EmptyCanTrackTOG(IN := sEmpty_Can_Track, RESET := NOT iEmergency_Stop); // TOGGLE
_w3 := (EmptyCanTrackTOG.Q OR CleanMode) AND iEmergency_Stop;
oEmpty_Can_Conv := _w3;
oEmpty_Can_Track := _w3;

// NETWORK 48
CloserSteamControl_Tog(IN := sCloserSteamEnable, RESET := FALSE); // TOGGLE
sCloserSteamEnable_Lt := CloserSteamControl_Tog.Q;

// NETWORK 49

// NETWORK 50
Closer_Steam_Low_Disable_Delay(IN := FALSE AND CloserSteamControl_Tog.Q AND oCloser AND NOT sCloser_Steam_ON, PT := T#5s); // TON
Closer_Steam_Low_Disable := Closer_Steam_Low_Disable_Delay.Q;

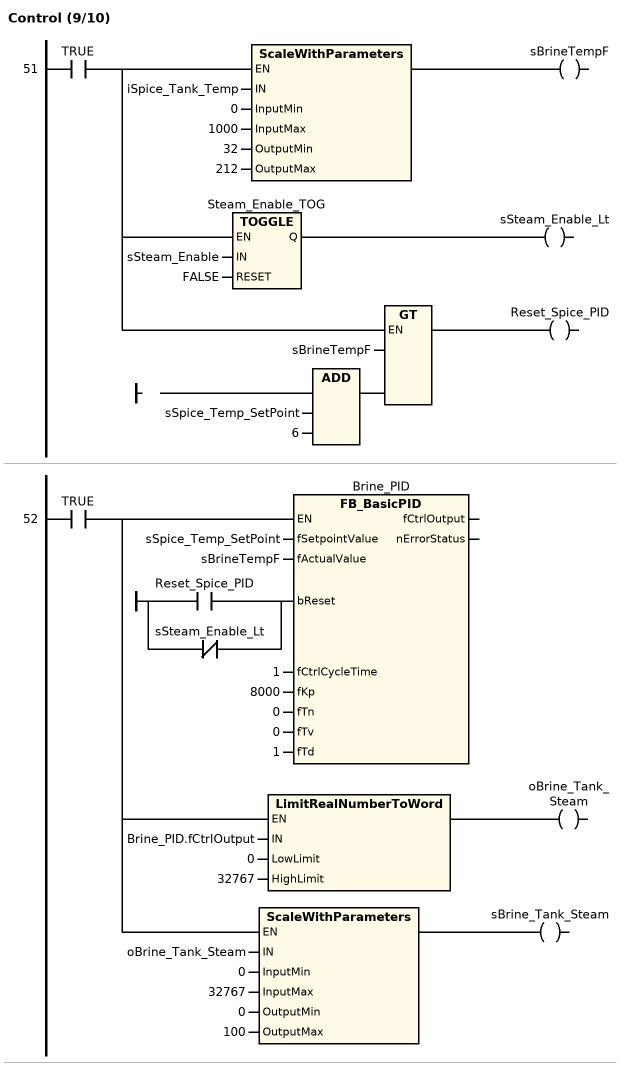
// NETWORK 51
sBrineTempF := ScaleWithParameters(IN := iSpice_Tank_Temp, InputMin := 0, InputMax := 1000, OutputMin := 32, OutputMax := 212);
Steam_Enable_TOG(IN := sSteam_Enable, RESET := FALSE); // TOGGLE
sSteam_Enable_Lt := Steam_Enable_TOG.Q;
Reset_Spice_PID := sBrineTempF > sSpice_Temp_SetPoint + 6;

// NETWORK 52
Brine_PID(
    fSetpointValue := sSpice_Temp_SetPoint,
    fActualValue := sBrineTempF,
    bReset := Reset_Spice_PID OR NOT sSteam_Enable_Lt,
    fCtrlCycleTime := 1,
    fKp := 8000,
    fTn := 0,
    fTv := 0,
    fTd := 1); // FB_BasicPID
oBrine_Tank_Steam := LimitRealNumberToWord(IN := Brine_PID.fCtrlOutput, LowLimit := 0, HighLimit := 32767);
sBrine_Tank_Steam := ScaleWithParameters(IN := oBrine_Tank_Steam, InputMin := 0, InputMax := 32767, OutputMin := 0, OutputMax := 100);

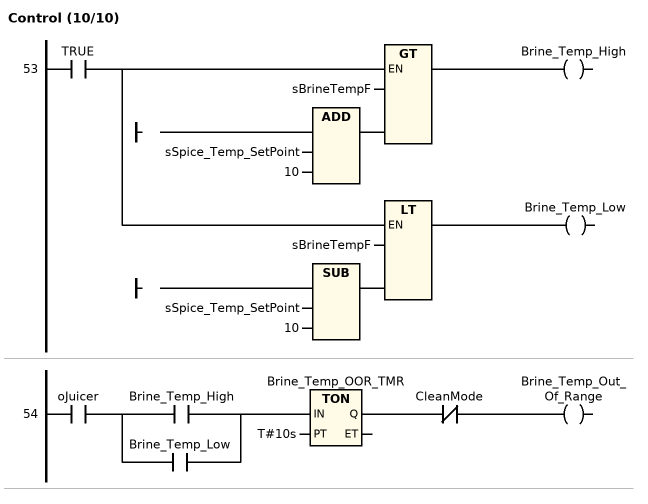
// NETWORK 53
Brine_Temp_High := sBrineTempF > sSpice_Temp_SetPoint + 10;
Brine_Temp_Low := sBrineTempF < sSpice_Temp_SetPoint - 10;

// NETWORK 54
Brine_Temp_OOR_TMR(IN := oJuicer AND (Brine_Temp_High OR Brine_Temp_Low), PT := T#10s); // TON
Brine_Temp_Out_Of_Range := Brine_Temp_OOR_TMR.Q AND NOT CleanMode;

END_PROGRAM

// ---- POUs/Hopper_Level.TcPOU
FUNCTION_BLOCK Hopper_Level
VAR_INPUT
	HopperLevel_Input:WORD;
END_VAR
VAR_OUTPUT
	HopperLevel_PCT:REAL;
END_VAR
VAR
	HopperLevel_Real: REAL;
END_VAR

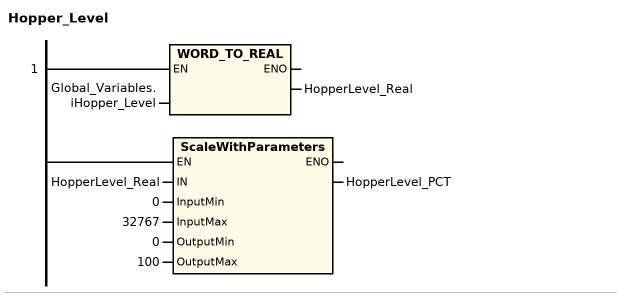
// NETWORK 1
HopperLevel_Real := WORD_TO_REAL(Global_Variables.iHopper_Level);
HopperLevel_PCT := ScaleWithParameters(IN := HopperLevel_Real, InputMin := 0, InputMax := 32767, OutputMin := 0, OutputMax := 100);

END_FUNCTION_BLOCK

// ---- POUs/Function Blocks/ScaleWithParameters.TcPOU
FUNCTION ScaleWithParameters : REAL
VAR_INPUT
	IN : REAL;
	InputMin : INT;
	InputMax : INT;
	OutputMin : REAL;
	OutputMax : REAL;
END_VAR
VAR
	InputSpan : INT;
	InputPercent : REAL;
	OutputSpan : REAL;
END_VAR

InputSpan := InputMax - InputMin;

(* Prevent divide by zero *)
IF InputSpan=0 THEN
	InputSpan:=1;
END_IF

OutputSpan := OutputMax - OutputMin;

InputPercent := (IN - InputMin) / INT_TO_REAL (InputSpan);

ScaleWithParameters := InputPercent * OutputSpan + OutputMin;

END_FUNCTION

// ---- POUs/Function Blocks/FillerCPM_Current.TcPOU
FUNCTION_BLOCK FillerCPM_Current
VAR_INPUT
	Filler_PulseInput : BOOL;
END_VAR
VAR_OUTPUT
	Current_Can_Pulses : REAL;
    CPM_Reading : REAL;
END_VAR
VAR
	fb_RisingEdge : R_TRIG;
    fb_MinuteTimer : TON;
    udiCurrentPulseCount : REAL := 0;
END_VAR

// Rising edge detection for pulse input
    fb_RisingEdge(CLK := Filler_PulseInput);
	IF fb_RisingEdge.Q THEN
        udiCurrentPulseCount := udiCurrentPulseCount + 1;
    END_IF
	// Minute timer
    fb_MinuteTimer(IN := TRUE, PT := T#20S); // Start timer automatically

    // When the minute timer expires
    IF fb_MinuteTimer.Q THEN
		
        // Store the current count as the last minute's count
        CPM_Reading := (udiCurrentPulseCount*3 * 0.75);
        // Reset the current pulse count for the new minute
        udiCurrentPulseCount := 0;
        // Reset the timer to start counting for the next minute
        fb_MinuteTimer(IN := FALSE); // Reset timer
        fb_MinuteTimer(IN := TRUE, PT := T#20S);//Restart timer
    END_IF

    // Output the current minute's pulse count
    Current_Can_Pulses := udiCurrentPulseCount;

END_FUNCTION_BLOCK

// ---- POUs/Function Blocks/LimitRealNumberToWord.TcPOU
FUNCTION LimitRealNumberToWord : INT
VAR_INPUT
	IN : REAL;
	LowLimit : REAL;
	HighLimit : REAL;
END_VAR
VAR
END_VAR

LimitRealNumberToWord:=REAL_TO_WORD(LimitRealNumber(IN,LowLimit,HighLimit));

END_FUNCTION

// ---- POUs/Function Blocks/LimitRealNumber.TcPOU
FUNCTION LimitRealNumber : REAL
VAR_INPUT
	IN : REAL;
	LowLimit : REAL;
	HighLimit : REAL;
END_VAR
VAR
END_VAR

LimitRealNumber:= IN;

IF (IN<LowLimit) THEN
	LimitRealNumber:= LowLimit;
END_IF

IF (IN>HighLimit) THEN
	LimitRealNumber:= HighLimit;
END_IF

END_FUNCTION

// ---- POUs/Messages.TcPOU
PROGRAM Messages
VAR

END_VAR

sMessages:='No Messages';

IF Jam_Fault THEN
sMessages:='Closer Area Jam!';
END_IF

IF NOT iEmergency_Stop THEN
sMessages:='Emergency Stop!';
END_IF

IF Low_Spice_Alarm THEN
	sMessages:='Low Level detected in SPICE TANK!!! ';
END_IF

IF Low_Spice_Disable THEN
	sMessages:='Line Paused....Low Level detected in SPICE TANK!!! ';
END_IF

IF Global_Variables_HMI.HopperLevel_IS_HIGH THEN
	sMessages:='High Level in Surge Hopper.....Infeed Auger Paused!!! ';
END_IF

IF Brine_Temp_Out_Of_Range THEN
	sMessages:='Brine Temp Out of Range!!!' ;
END_IF

IF Closer_Steam_Low_Disable THEN
	sMessages:='Line Paused Due To Low Steam at Closer!';
END_IF

IF Global_Variables_HMI.HopperLevelIS_LOW THEN
	sMessages:='Low Level in Surge Hopper.....Infeed Auger Paused!!! ';
END_IF

END_PROGRAM

// ---- POUs/Speed_Setpoints.TcPOU
PROGRAM Speed_Setpoints
VAR

	oSpicePumpSpeed: REAL;

	oCloserSpeed: REAL;
	Spare1Setpoint: INT;
	Spare2Setpoint: INT;

	Sp1: INT;
	Sp2: INT;

	Exit_Conv_Speed_SPt: INT;
	test: REAL;
	Spiral_Infeed_Spt: INT;
	Spiral_Infeed_Setpoint: INT;

END_VAR
VAR // added by the converter: edge detectors and wires of the graphical bodies
    _w1, _w2 : ANY;
END_VAR

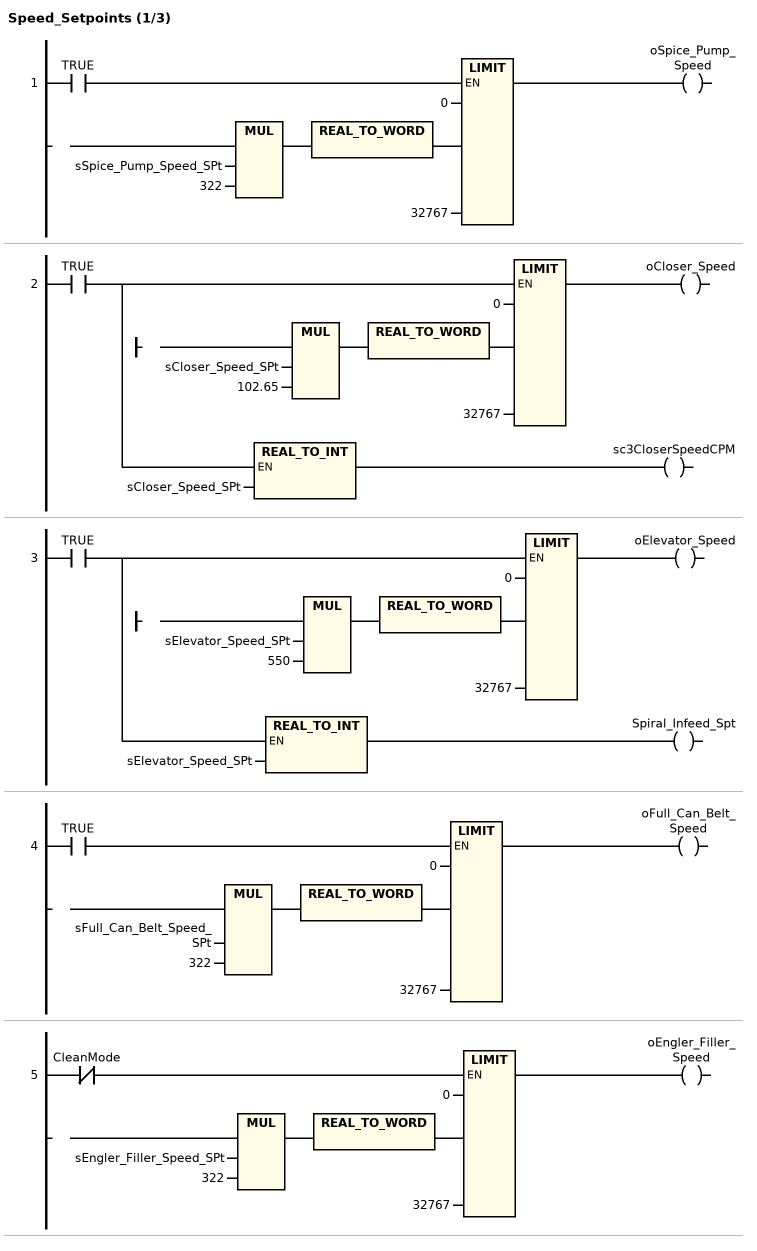
// NETWORK 1
oSpice_Pump_Speed := LIMIT(0, REAL_TO_WORD(sSpice_Pump_Speed_SPt * 322), 32767);

// NETWORK 2
oCloser_Speed := LIMIT(0, REAL_TO_WORD(sCloser_Speed_SPt * 102.65), 32767);
sc3CloserSpeedCPM := REAL_TO_INT(sCloser_Speed_SPt);

// NETWORK 3
oElevator_Speed := LIMIT(0, REAL_TO_WORD(sElevator_Speed_SPt * 550), 32767);
Spiral_Infeed_Spt := REAL_TO_INT(sElevator_Speed_SPt);

// NETWORK 4
oFull_Can_Belt_Speed := LIMIT(0, REAL_TO_WORD(sFull_Can_Belt_Speed_SPt * 322), 32767);

// NETWORK 5
IF NOT CleanMode THEN _w1 := LIMIT(0, REAL_TO_WORD(sEngler_Filler_Speed_SPt * 322), 32767); END_IF
oEngler_Filler_Speed := _w1;

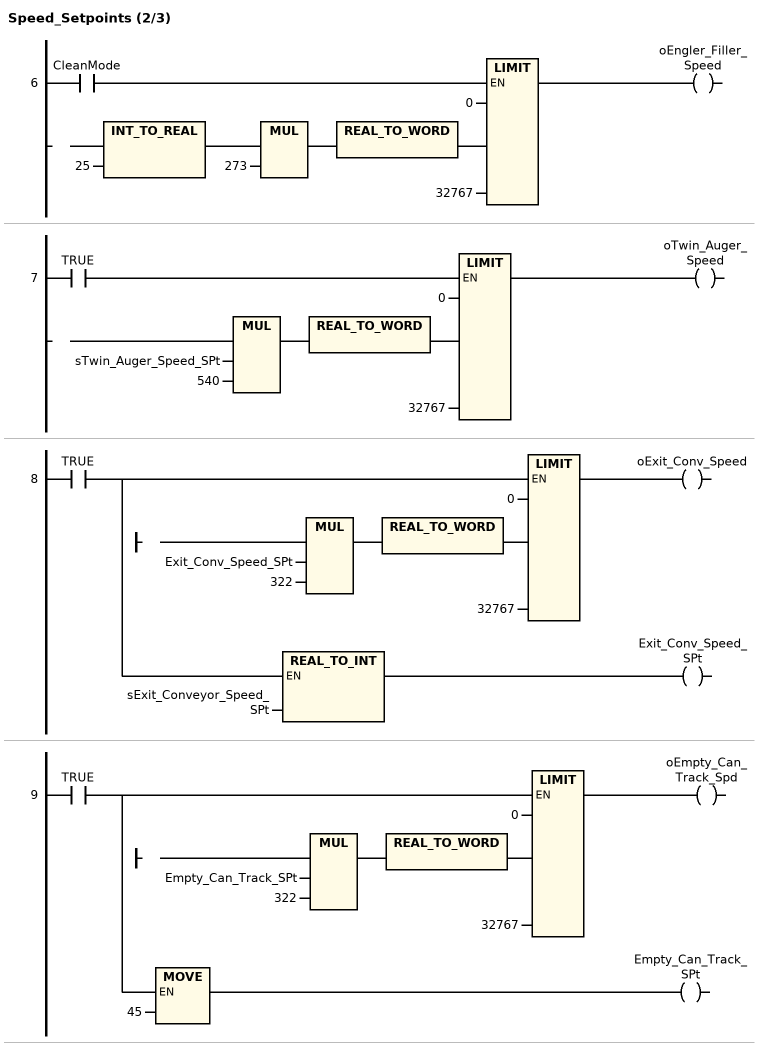
// NETWORK 6
IF CleanMode THEN _w2 := LIMIT(0, REAL_TO_WORD(INT_TO_REAL(25) * 273), 32767); END_IF
oEngler_Filler_Speed := _w2;

// NETWORK 7
oTwin_Auger_Speed := LIMIT(0, REAL_TO_WORD(sTwin_Auger_Speed_SPt * 540), 32767);

// NETWORK 8
oExit_Conv_Speed := LIMIT(0, REAL_TO_WORD(Exit_Conv_Speed_SPt * 322), 32767);
Exit_Conv_Speed_SPt := REAL_TO_INT(sExit_Conveyor_Speed_SPt);

// NETWORK 9
oEmpty_Can_Track_Spd := LIMIT(0, REAL_TO_WORD(Empty_Can_Track_SPt * 322), 32767);
Empty_Can_Track_SPt := 45;

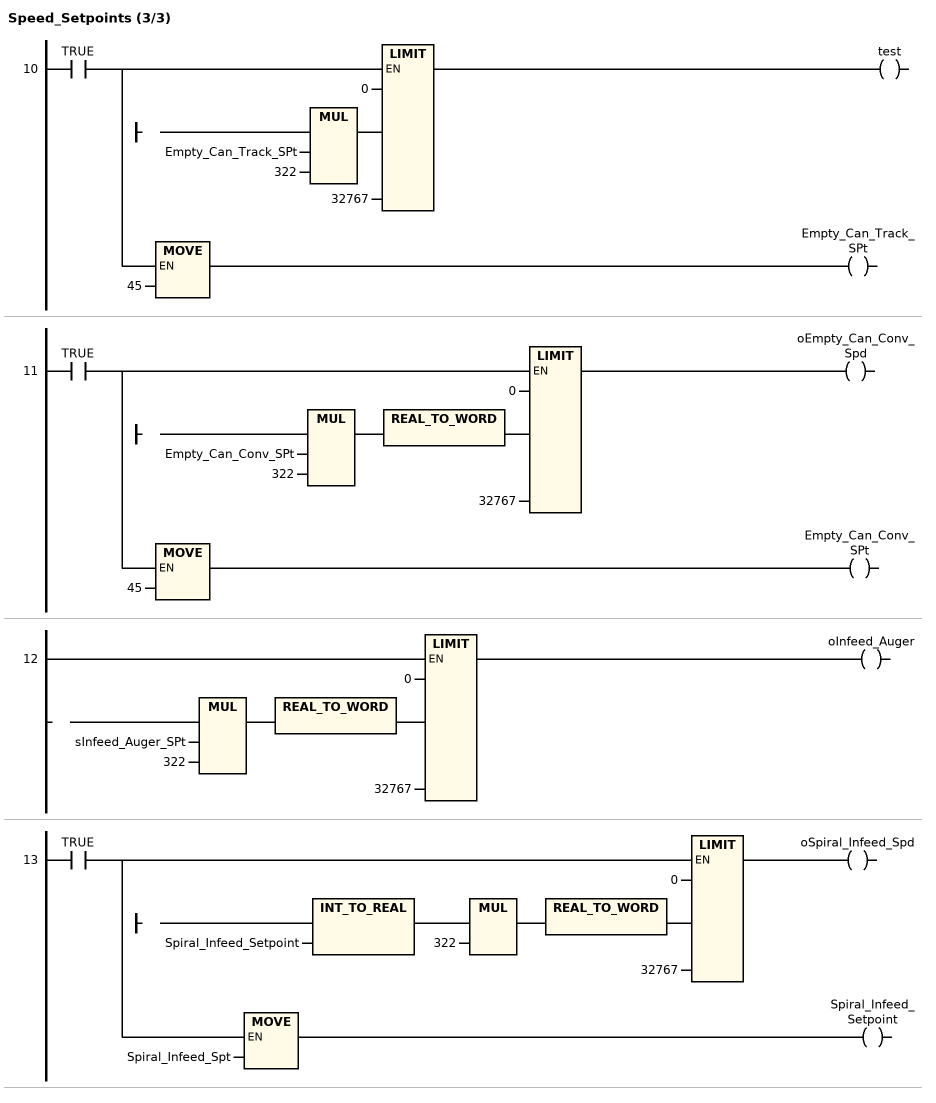
// NETWORK 10
test := LIMIT(0, Empty_Can_Track_SPt * 322, 32767);
Empty_Can_Track_SPt := 45;

// NETWORK 11
oEmpty_Can_Conv_Spd := LIMIT(0, REAL_TO_WORD(Empty_Can_Conv_SPt * 322), 32767);
Empty_Can_Conv_SPt := 45;

// NETWORK 12
oInfeed_Auger := LIMIT(0, REAL_TO_WORD(sInfeed_Auger_SPt * 322), 32767);

// NETWORK 13
oSpiral_Infeed_Spd := LIMIT(0, REAL_TO_WORD(INT_TO_REAL(Spiral_Infeed_Setpoint) * 322), 32767);
Spiral_Infeed_Setpoint := Spiral_Infeed_Spt;

END_PROGRAM

// ---- POUs/StandardCPM.TcPOU
PROGRAM StandardCPM
VAR
	ProdStd : REAL;
	BriteCode_Standards : StandardCPMSet;
END_VAR

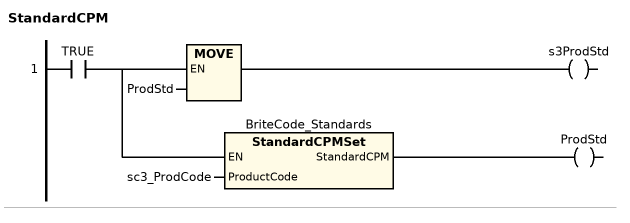
// NETWORK 1
s3ProdStd := ProdStd;
BriteCode_Standards(ProductCode := sc3_ProdCode); // StandardCPMSet
ProdStd := BriteCode_Standards.StandardCPM;

END_PROGRAM

// ---- POUs/Function Blocks/StandardCPMSet.TcPOU
FUNCTION_BLOCK StandardCPMSet
VAR_INPUT
	ProductCode : STRING;

END_VAR
VAR_OUTPUT
	StandardCPM: REAL;

END_VAR
VAR

END_VAR

IF ProductCode='2BEBACBBB - 300 Brite Blackeye w/Bacon'  THEN StandardCPM:=294; END_IF
IF ProductCode='2BEBBB - 300 Brite Blackeye Peas'  THEN StandardCPM:=294; END_IF
IF ProductCode='2BEBACBBB - 300 Brite Trappeys Blkeye/Jalapeno/Bacon'  THEN StandardCPM:=294; END_IF
IF ProductCode='2BKBBB - 300 Brite Black Beans Salt/Water'  THEN StandardCPM:=294; END_IF
IF ProductCode='2BKFBBB - 300 Brite Black Beans Fully Seas'  THEN StandardCPM:=294; END_IF
IF ProductCode='2BPBBB - 300 Brite Butter Peas'  THEN StandardCPM:=294; END_IF
IF ProductCode='2CBBBB - 300 Brite Spiced Chili Beans'  THEN StandardCPM:=294; END_IF
IF ProductCode='2CPBMFBBB - 300 Brite Cajun Pinto Beans'  THEN StandardCPM:=294; END_IF
IF ProductCode='2CRBBB - 300 Brite Crowder Peas'  THEN StandardCPM:=294; END_IF
IF ProductCode='2FPBACBBB - 300 Brite Trappey FP W/ Bacon'  THEN StandardCPM:=294; END_IF
IF ProductCode='2FPBBB - 300 Brite Field Peas CR'  THEN StandardCPM:=294; END_IF
IF ProductCode='2FPSBACBBB - 300 Brite Trappey FP W/ Bacon & Snaps'  THEN StandardCPM:=294; END_IF
IF ProductCode='2FPSBBB - 300 Brite Field Peas/Snaps CR'  THEN StandardCPM:=294; END_IF
IF ProductCode='2GLSBEBB - 300 Brite Glory Sen Seas Blackeyes'  THEN StandardCPM:=294; END_IF
IF ProductCode='2GSBBBBB - 300 Brite Glory Seas Butter Beans'  THEN StandardCPM:=294; END_IF
IF ProductCode='2GSBEBBB - 300 Brite Glory Seas Blackeyes'  THEN StandardCPM:=294; END_IF
IF ProductCode='2GSFPSBB - 300 Brite Glory Seas Field Peas/Snaps CR'  THEN StandardCPM:=294; END_IF
IF ProductCode='2GSLBBBB - 300 Brite Glory Seas Lima Beans'  THEN StandardCPM:=294; END_IF
IF ProductCode='2GSNOBBB - 300 Brite Glory Seas Northern Beans'  THEN StandardCPM:=294; END_IF
IF ProductCode='2GSPBBBB - 300 Brite Glory Seas Pinto Beans'  THEN StandardCPM:=294; END_IF
IF ProductCode='2GSPBOBB - 300 Brite Glory Seas Pinto Beans/Onions'  THEN StandardCPM:=294; END_IF
IF ProductCode='2GVBEBB - 300 Brite Great Value Blackeye Peas'  THEN StandardCPM:=294; END_IF
IF ProductCode='2LBBACBB - 300 Brite Trappey  Lima Bean with Bacon'  THEN StandardCPM:=294; END_IF
IF ProductCode='2LBBBB - 300 Brite Medium Green Lima Beans'  THEN StandardCPM:=294; END_IF
IF ProductCode='2LGBBB - 300 Brite Large Lima Beans'  THEN StandardCPM:=294; END_IF
IF ProductCode='2LKBBBB - 300 Brite Light Kidney Beans'  THEN StandardCPM:=294; END_IF
IF ProductCode='2LSBEBBB - 300 Brite Low Sodium Blackeye Peas'  THEN StandardCPM:=294; END_IF
IF ProductCode='2LSBKBBB - 300 Brite Low Sod Black Beans S&W'  THEN StandardCPM:=294; END_IF
IF ProductCode='2LSDRKGBBB - 300 Brite Low Sod Dark Kidney Beans'  THEN StandardCPM:=294; END_IF
IF ProductCode='2LSGBKBBB - 300 Brite Low Sod Govt Black Beans'  THEN StandardCPM:=294; END_IF
IF ProductCode='2MBNBBB - 300 Brite Mixed Beans'  THEN StandardCPM:=294; END_IF
IF ProductCode='2NBACBBB - 300 Brite Trappey  Navy Bean with Bacon'  THEN StandardCPM:=294; END_IF
IF ProductCode='2NBBBB - 300 Brite Navy Beans'  THEN StandardCPM:=294; END_IF
IF ProductCode='2NJBACBBB - 300 Brite Navy Bean/Jalapeno/Bacon'  THEN StandardCPM:=294; END_IF
IF ProductCode='2RSGSLBB - 300 Brite Glory Med Grn Limas Red Sodium'  THEN StandardCPM:=294; END_IF
IF ProductCode='2NOBBBB - 300 Brite Great Northern Beans'  THEN StandardCPM:=294; END_IF
IF ProductCode='2NOSKBBB - 300 Trappeys Lt Red Kidney Bns NO Seas'  THEN StandardCPM:=294; END_IF
IF ProductCode='2PBBACBBB - 300 Brite Trappey Pinto Beans with Bacon'  THEN StandardCPM:=294; END_IF
IF ProductCode='2PBBBB - 300 Brite Pinto Beans'  THEN StandardCPM:=294; END_IF
IF ProductCode='2PBJBACBBB - 300 Brite Trappey Pinto w/Jalapeno/Bacon'  THEN StandardCPM:=294; END_IF
IF ProductCode='2PPBBB - 300 Brite Pepper N Peas CR'  THEN StandardCPM:=294; END_IF
IF ProductCode='2RKCHBBB - 300 Brite Red Kidney Beans with Chili'  THEN StandardCPM:=294; END_IF
IF ProductCode='2RSGSBEB - 300 Brite Glory Blackeye Peas Red Sodium'  THEN StandardCPM:=294; END_IF
IF ProductCode='2RSGSFPSB - 300 Brite Glry Red Sod FP/Snaps'  THEN StandardCPM:=294; END_IF
IF ProductCode='2SBEBBB - 300 Brite Seas Blackeyes'  THEN StandardCPM:=294; END_IF
IF ProductCode='2SFSBBB - 300 Brite Seas Fld Peas/Snaps CR'  THEN StandardCPM:=294; END_IF
IF ProductCode='2SLBBBB - 300 Brite Seas Medium Green Limas'  THEN StandardCPM:=294; END_IF
IF ProductCode='2SLGBBB - 300 Brite Seas Butterbeans'  THEN StandardCPM:=294; END_IF
IF ProductCode='2SPBBBB - 300 Brite Seas Pinto Beans'  THEN StandardCPM:=294; END_IF
IF ProductCode='2WABBB - 300 Brite White Acre Peas'  THEN StandardCPM:=294; END_IF
IF ProductCode='2GLSCGBB - 300 Brite Glory Sen Seas Collard Greens'  THEN StandardCPM:=172; END_IF
IF ProductCode='2GLSMGBB - 300 Brite Glory Sen Seas Mixed Greens'  THEN StandardCPM:=172; END_IF
IF ProductCode='2GLSTGBB - 300 Brite Glory Sen Seas Turnips'  THEN StandardCPM:=172; END_IF
IF ProductCode='2GSTCGBB - 300 Brite Glory Seas Smk Turkey Collards'  THEN StandardCPM:=172; END_IF
IF ProductCode='2GSTMGBB - 300 Brite Glory Turkey Mixed Greens'  THEN StandardCPM:=172; END_IF
IF ProductCode='2GSTTGBB - 300 Brite Glory Seas Smk Turkey Turnips'  THEN StandardCPM:=172; END_IF
IF ProductCode='2GVCGBB - 300 Brite Great Value Collard Greens'  THEN StandardCPM:=172; END_IF
IF ProductCode='2GVTGBB - 300 Brite GV Turnip Greens'  THEN StandardCPM:=172; END_IF
IF ProductCode='2NCGBBB - 300 Brite No-Salt Collard Greens Chopped'  THEN StandardCPM:=172; END_IF
IF ProductCode='2NKABBB - 300 Brite No Salt Kale Greens Chopped'  THEN StandardCPM:=172; END_IF
IF ProductCode='2NMGBBB - 300 Brite No-Salt Mixed Greens Chopped'  THEN StandardCPM:=172; END_IF
IF ProductCode='2NMUBBB - 300 Brite No-Salt Mustard Greens Chopped'  THEN StandardCPM:=172; END_IF
IF ProductCode='2NTGBBB - 300 Brite No-Salt Turnip Greens Chopped'  THEN StandardCPM:=172; END_IF
IF ProductCode='2NTWBBB - 300 Brite No-Salt Turnip/Roots Chopped'  THEN StandardCPM:=172; END_IF
IF ProductCode='2RSGSCGB - 300 Brite Glory Red Sodium Collard Grns'  THEN StandardCPM:=172; END_IF
IF ProductCode='2RSGSMGB - 300 Brite Glory Mixed Greens Red Sodium'  THEN StandardCPM:=172; END_IF
IF ProductCode='2RSGSTGB - 300 Brite Glory Red Sodium Turnip Grns'  THEN StandardCPM:=172; END_IF
IF ProductCode='2SCGBBB - 300 Brite Seas Collard Greens'  THEN StandardCPM:=172; END_IF
IF ProductCode='2SMGBBB - 300 Brite Seas Mixed Greens'  THEN StandardCPM:=172; END_IF
IF ProductCode='2SMUBBB - 300 Brite Seas Mustard Greens'  THEN StandardCPM:=172; END_IF
IF ProductCode='2STGBBB - 300 Brite Seas Turnips'  THEN StandardCPM:=172; END_IF
IF ProductCode='2STWBBB - 300 Brite Seas Turnip/Roots'  THEN StandardCPM:=172; END_IF
IF ProductCode='2BNDMBBB - 300 Brite Allens Green Beans'  THEN StandardCPM:=130; END_IF
IF ProductCode='2BNSOBBB - 300 Shell Out Green Beans w-Pintos'  THEN StandardCPM:=130; END_IF
IF ProductCode='2FLNBNBBB - 300 Brite Freshlike NSA Green Beans'  THEN StandardCPM:=130; END_IF
IF ProductCode='2GLSBNBB - 300 Brite Glory Sen Seas Green Beans'  THEN StandardCPM:=130; END_IF
IF ProductCode='2GSBNBBB - 300 Brite Glory Seasoned Green Beans'  THEN StandardCPM:=130; END_IF
IF ProductCode='2ITBBBB - 300 Brite Italian Green Beans'  THEN StandardCPM:=130; END_IF
IF ProductCode='2ITBSOBBB - 300 Brite Shell Out Italian Beans w-Pint'  THEN StandardCPM:=130; END_IF
IF ProductCode='2LSBNBBB - 300 Brite Low Sodium Green Beans'  THEN StandardCPM:=130; END_IF
IF ProductCode='2RSGSBNB - 300 Brite Glory Red Sodium Seas Grn Bean'  THEN StandardCPM:=130; END_IF
IF ProductCode='2SITBBB - 300 Brite Seasoned Italian Green Beans'  THEN StandardCPM:=130; END_IF
IF ProductCode='2HOMCWBBB - 300 Brite White Cracked Hominy'  THEN StandardCPM:=240; END_IF
IF ProductCode='2HOMGBBB - 300 Brite Golden Hominy'  THEN StandardCPM:=240; END_IF
IF ProductCode='2HOMGEZOB - 300 Brite Golden Hominy-EZO'  THEN StandardCPM:=240; END_IF
IF ProductCode='2HOMWBBB - 300 Brite White Hominy'  THEN StandardCPM:=240; END_IF
IF ProductCode='2HOMWEZOB - 300 Brite White Hominy-EZO'  THEN StandardCPM:=240; END_IF
IF ProductCode='2LSHOMWBB - 300 Brite LS White Hominy'  THEN StandardCPM:=240; END_IF
IF ProductCode='2BCORBBB - 300 Brite Buttered Corn'  THEN StandardCPM:=155; END_IF
IF ProductCode='2BSUCBBB - 300 Brite Double Succotash'  THEN StandardCPM:=155; END_IF
IF ProductCode='2BUFPNBBB - 300 Brite Buffalo Peanuts'  THEN StandardCPM:=180; END_IF
IF ProductCode='2CPNBBB - 300 Brite Cajun Boiled Peanuts'  THEN StandardCPM:=180; END_IF
IF ProductCode='2DLPNBBB - 300 Brite Dill Peanuts'  THEN StandardCPM:=180; END_IF
IF ProductCode='2HOTPNBBB - 300 Brite Hot Sauce Peanuts'  THEN StandardCPM:=180; END_IF
IF ProductCode='2JALPNBBB - 300 Brite Jalapeno Peanuts'  THEN StandardCPM:=180; END_IF
IF ProductCode='2PNBBB - 300 Brite Boiled Peanuts'  THEN StandardCPM:=180; END_IF
IF ProductCode='2SPDLPNBBB - 300 Brite Spicy Dill Peanuts'  THEN StandardCPM:=180; END_IF
IF ProductCode='2SVPNBB - 300 Brite Salt/Vinegar Boiled Peanuts'  THEN StandardCPM:=180; END_IF
IF ProductCode='2GLSTOBB - 300 Brite Glory Sen Seas Tom & Okra'  THEN StandardCPM:=260; END_IF
IF ProductCode='2GLSTOCB - 300 Brite Glory Sen Seas Tom/Okra/ Corn'  THEN StandardCPM:=260; END_IF
IF ProductCode='2HJBBB - 300 Brite Hoppin John'  THEN StandardCPM:=260; END_IF
IF ProductCode='2RSTOBB - 300 Brite Glory Red Sodium Tom & Okra'  THEN StandardCPM:=260; END_IF
IF ProductCode='2RSTOCBB - 300 Brite Glory Red SodiumTom/Okra/ Corn'  THEN StandardCPM:=260; END_IF
IF ProductCode='2SUCBBB - 300 Brite Succotash/Triple'  THEN StandardCPM:=260; END_IF
IF ProductCode='2TOBBB - 300 Brite Tomatoes/Okra'  THEN StandardCPM:=260; END_IF
IF ProductCode='2TOCBBB - 300 Brite Tomatoes/Okra/Corn'  THEN StandardCPM:=260; END_IF
IF ProductCode='2COGUMBB - 300 Brite Creole Okra Gumbo'  THEN StandardCPM:=160; END_IF
IF ProductCode='2LSVAMVBBB - 300 Brite Low Sodium Mixed Vegetables'  THEN StandardCPM:=160; END_IF
IF ProductCode='2LSVAMVGBBB - 300 Brite Low Sodium Veg All - All DC'  THEN StandardCPM:=160; END_IF
IF ProductCode='2NVAMVBBB - 300 Brite Veg-All Mixed Vegetables NSA'  THEN StandardCPM:=160; END_IF
IF ProductCode='2OKBBB - 300 Brite Cut Okra'  THEN StandardCPM:=160; END_IF
IF ProductCode='2RSCOGUMB - 300 Brite Creole Okra Gumbo Red Sodium'  THEN StandardCPM:=160; END_IF
IF ProductCode='2VAMVBBB - 300 Brite Veg-All Mixed Vegetables'  THEN StandardCPM:=160; END_IF
IF ProductCode='2LSSIBBB - 300 Brite Spinach LS Cut Leaf ¾" x ¾"'  THEN StandardCPM:=145; END_IF
IF ProductCode='2LSSIGBB - 300 Brite Low Sodium Spinach-G-NA'  THEN StandardCPM:=145; END_IF
IF ProductCode='2NSIBBB - 300 Brite Spinach NSA Cut Leaf ¾" x ¾"'  THEN StandardCPM:=145; END_IF
IF ProductCode='2SIBBB - 300 Brite Spinach Cut Leaf 3/4" x 3/4"'  THEN StandardCPM:=145; END_IF
IF ProductCode='2SICHBBB - 300 Brite Spinach Chopped ½" x ½"'  THEN StandardCPM:=145; END_IF
IF ProductCode='2SIPTBB - 300 Brite Spinach - EZO'  THEN StandardCPM:=145; END_IF
IF ProductCode='2RSGSIB - 300 Glory Spinach Reduced Sodium'  THEN StandardCPM:=145; END_IF
IF ProductCode='2YCANDBB - 300 Brite Candied Yams'  THEN StandardCPM:=120; END_IF
IF ProductCode='2YCUTBBB - 300 Brite Cut Yams'  THEN StandardCPM:=120; END_IF
IF ProductCode='2YCUTELSBBB - 300 Brite Extra Light Syrup Cut Yams'  THEN StandardCPM:=120; END_IF
IF ProductCode='2YCUTELSC1BBB - 300 Brite Extra Light Syrup Yams-3PC'  THEN StandardCPM:=120; END_IF
IF ProductCode='2YOPBBB - 300 Brite Yams in Orange/Pineapple Sauce'  THEN StandardCPM:=120; END_IF
IF ProductCode='2SQBBB - 300 Brite Yellow Squash Cut'  THEN StandardCPM:=140; END_IF
IF ProductCode='2SQOBBB - 300 Brite Squash & Onions'  THEN StandardCPM:=140; END_IF
IF ProductCode='2GSCABBB - 300 Brite Glory Country Style Cabbage'  THEN StandardCPM:=195; END_IF
IF ProductCode='2SCABBB - 300 Brite Seas Cabbage'  THEN StandardCPM:=195; END_IF
IF ProductCode='2GSCORBBB - 300 Brite Glory Skillet Corn'  THEN StandardCPM:=128; END_IF
IF ProductCode='2RSGSCORB - 300 Brite Glry Skillet Reduce SodiumCorn'  THEN StandardCPM:=128; END_IF
IF ProductCode='4HOMGBBB - 2.5 Brite Golden Hominy'  THEN StandardCPM:=128; END_IF
IF ProductCode='4HOMWBBB - 2.5 Brite White Hominy'  THEN StandardCPM:=128; END_IF
IF ProductCode='2GFABBB - 300 Brite Glory Fried Apples'  THEN StandardCPM:=164; END_IF
IF ProductCode='2MHFABBB - 300 Brite MH Fried Apples'  THEN StandardCPM:=164; END_IF
IF ProductCode='2RSGHCARB - 300 Brite Glory Honey Carrots Red Sodium'  THEN StandardCPM:=206; END_IF
IF ProductCode='2RUTBBB - 300 Brite Rutabagas'  THEN StandardCPM:=206; END_IF
IF ProductCode='2GHCARBB - 300 Brite Glory Honey Carrots'  THEN StandardCPM:=206; END_IF
IF ProductCode='2GSBERBB - 300 Brite Glory Seas Blackeyes & Rice'  THEN StandardCPM:=244; END_IF
IF ProductCode='2GSRBRBB - 300 Brite Glory Seas Red Beans/Rice'  THEN StandardCPM:=244; END_IF
IF ProductCode='2RBRBBB - 300 Brite Red Beans/Rice'  THEN StandardCPM:=244; END_IF
IF ProductCode='40BNBBB - 40oz Brite Blue Lake Green Beans'  THEN StandardCPM:=80; END_IF
IF ProductCode='40BNPBBB - 40oz Brite Blue Lake Green Bean/Potatoes'  THEN StandardCPM:=80; END_IF
IF ProductCode='40ITBBBB - 38oz Brite Italian Green Beans'  THEN StandardCPM:=80; END_IF
IF ProductCode='40SBNBBB - 40oz Brite Blue Lake Seas Green Beans'  THEN StandardCPM:=80; END_IF
IF ProductCode='40YCTELSBBB - 40oz Brite Extra Light Syrup Cut Yams'  THEN StandardCPM:=110; END_IF
IF ProductCode='40YCTSFBB - 40oz Bruce Yams Sugar Free'  THEN StandardCPM:=110; END_IF
IF ProductCode='40YMPBBB - 40 oz Brite Princella Cut Sweet Pot NSA'  THEN StandardCPM:=110; END_IF
IF ProductCode='4ALSITBBB - 2.5 Brite Allens Seas Ital Beans'  THEN StandardCPM:=110; END_IF
IF ProductCode='4BNBBB - 2.5 Brite Cut Green Beans'  THEN StandardCPM:=110; END_IF
IF ProductCode='4GSBNBBB - 2.5 Brite Glory Seas Green Beans'  THEN StandardCPM:=110; END_IF
IF ProductCode='4GSBNPBB - 2.5 Brite Glory Seas Green Bns/Potatoes'  THEN StandardCPM:=110; END_IF
IF ProductCode='4ITBBB - 2.5 Brite Italian Green Beans'  THEN StandardCPM:=110; END_IF
IF ProductCode='4SITBBB - 2.5 Brite Seas Ital Grn Bns'  THEN StandardCPM:=110; END_IF
IF ProductCode='4YCTSFBB - 2.5 Brite Cut Yams Sugar Free'  THEN StandardCPM:=110; END_IF
IF ProductCode='4YCUTBBB - 2.5 Brite Cut Yams'  THEN StandardCPM:=110; END_IF
IF ProductCode='4YCUTELSBBB - 2.5 Brite Extra Light Syrup Cut Yams'  THEN StandardCPM:=110; END_IF
IF ProductCode='4YGFCANBBB - 2.5 Brite Glory Candied Yams'  THEN StandardCPM:=110; END_IF
IF ProductCode='4BQPNBBB - 2.5 Brite Boiled Hot and Spicy Peanuts'  THEN StandardCPM:=125; END_IF
IF ProductCode='4BUFPNBBB - 2.5 Brite Buffalo Peanuts'  THEN StandardCPM:=125; END_IF
IF ProductCode='4DBUFPNBB - 2.5 Brite Dry Spicy Buffalo Peanuts'  THEN StandardCPM:=125; END_IF
IF ProductCode='4DLPNBBB - 2.5 Brite Dill Peanuts'  THEN StandardCPM:=125; END_IF
IF ProductCode='4GSCGBFB - 2.5 Brite Glory Seas FatBK Collard Green'  THEN StandardCPM:=124; END_IF
IF ProductCode='4GSKABFB - 2.5 Brite Glory Seas FatBK Kale Greens'  THEN StandardCPM:=124; END_IF
IF ProductCode='4GSMGBFB - 2.5 Brite Glory Seas FatBK Mixed Greens'  THEN StandardCPM:=124; END_IF
IF ProductCode='4GSMUBFB - 2.5 Brite Glory Seas FatBK Mustard Green'  THEN StandardCPM:=124; END_IF
IF ProductCode='4GSTGBFB - 2.5 Brite Glory Seas FatBK Turnip Greens'  THEN StandardCPM:=124; END_IF
IF ProductCode='4GSTWBFB - 2.5 Brite Glory Seas FatBK Turnips/Roots'  THEN StandardCPM:=124; END_IF
IF ProductCode='4HSMVBBB - 2.5 Brite Homestyle Mixed Vegetables'  THEN StandardCPM:=124; END_IF
IF ProductCode='4NTGBBB - 2.5 Brite NS Turnip Greens'  THEN StandardCPM:=124; END_IF
IF ProductCode='4PNBBB - 2.5 Brite Boiled Peanuts'  THEN StandardCPM:=124; END_IF
IF ProductCode='4SCGBBB - 2.5 Brite Seas Collard Greens'  THEN StandardCPM:=124; END_IF
IF ProductCode='4SMGBBB - 2.5 Brite Seas Mixed Greens'  THEN StandardCPM:=124; END_IF
IF ProductCode='4SMUBBB - 2.5 Brite Seas Mustard Greens'  THEN StandardCPM:=124; END_IF
IF ProductCode='4SPDLPNBBB - 2.5 Brite Spicy Dill Peanuts'  THEN StandardCPM:=124; END_IF
IF ProductCode='4STGBBB - 2.5 Brite Seas Turnip Greens'  THEN StandardCPM:=124; END_IF
IF ProductCode='4STWBBB - 2.5 Brite Seas Turnip/Roots'  THEN StandardCPM:=124; END_IF
IF ProductCode='4SVPNBB - 2.5 Brite Salt/Vinegar Boiled Peanuts'  THEN StandardCPM:=124; END_IF
IF ProductCode='4VAMVBBB - 2.5 Brite Veg-All Mixed Vegetables'  THEN StandardCPM:=124; END_IF
IF ProductCode='4SBBOBBB - 2.5 Brite S.Butter Bean w/Vid Onions'  THEN StandardCPM:=136; END_IF
IF ProductCode='4SBPOBBB - 2.5 Brite Seas Beans/Pot/Onion'  THEN StandardCPM:=136; END_IF
IF ProductCode='4SFPSOBBB - 2.5 Brite S. FP&Snaps w/VidOn CR'  THEN StandardCPM:=136; END_IF
IF ProductCode='4SPBOBBB - 2.5 Brite S. Pinto Bean w/Vid Onoions'  THEN StandardCPM:=136; END_IF
IF ProductCode='4CPBMFBBB - 2.5 Brite Cajun Pinto Beans'  THEN StandardCPM:=131; END_IF
IF ProductCode='4GSIBBB - 2.5 Brite Glory Seas Spinach'  THEN StandardCPM:=106; END_IF
IF ProductCode='4SIBBB - 2.5 Brite Spinach'  THEN StandardCPM:=106; END_IF
IF ProductCode='5ALCARDIBBB - #10 Brite Allens Diced Carrots'  THEN StandardCPM:=36; END_IF
IF ProductCode='5CPNBBB - #10 Brite Cajun Boiled Peanuts'  THEN StandardCPM:=45; END_IF
IF ProductCode='5DCPNBB - #10 Brite Dry Cajun Peanuts'  THEN StandardCPM:=45; END_IF
IF ProductCode='5HOMGBBB - #10 Brite Golden Hominy'  THEN StandardCPM:=45; END_IF
IF ProductCode='5HOMWBBB - #10 Brite White Hominy'  THEN StandardCPM:=45; END_IF
IF ProductCode='5HOMWJAUBBB - #10 Brite Mexican Hominy Juanita'  THEN StandardCPM:=45; END_IF
IF ProductCode='5HOMWSNBBB - #10 Brite Seneca White Hominy'  THEN StandardCPM:=45; END_IF
IF ProductCode='5ALCHHTBNBBB - #10 Brite Allens Chili Hot Beans'  THEN StandardCPM:=41; END_IF
IF ProductCode='5BCHBBB - #10 Brite Brooks Chili Hot Beans'  THEN StandardCPM:=41; END_IF
IF ProductCode='5BESBBB - #10 Brite Blackeye Peas/Snaps'  THEN StandardCPM:=41; END_IF
IF ProductCode='5BKFBBB - #10 Brite Black Beans Fully Seas'  THEN StandardCPM:=41; END_IF
IF ProductCode='5BONBBB - #10 Brite Garbanzo Beans'  THEN StandardCPM:=41; END_IF
IF ProductCode='5CHBRBB - #10 Brite Chili Beans w-Red Beans'  THEN StandardCPM:=41; END_IF
IF ProductCode='5CRBBB - #10 Brite Crowder Peas'  THEN StandardCPM:=41; END_IF
IF ProductCode='5FPBBB - #10 Brite Field Peas CR'  THEN StandardCPM:=41; END_IF
IF ProductCode='5FPSBBB - #10 Brite Field Peas/Snaps CR'  THEN StandardCPM:=41; END_IF
IF ProductCode='5LGBBB - #10 Brite Large Lima Beans'  THEN StandardCPM:=41; END_IF
IF ProductCode='5LKBBBB - #10 Brite Light Kidney Beans'  THEN StandardCPM:=41; END_IF
IF ProductCode='5LSBEBBB - #10 Brite Low Sodium Blackeye Peas'  THEN StandardCPM:=41; END_IF
IF ProductCode='5LSBKBBB - #10 Brite Low Sod Black Beans S&W'  THEN StandardCPM:=41; END_IF
IF ProductCode='5LSBKSCBB - #10 Brite LS Black Beans Slow Cook'  THEN StandardCPM:=41; END_IF
IF ProductCode='5LSKBBBB - #10 Brite Low Sodium Dark Kidney Beans'  THEN StandardCPM:=41; END_IF
IF ProductCode='5LSLBBBB - #10 Brite Low Sod Medium Green Limas'  THEN StandardCPM:=41; END_IF
IF ProductCode='5LSNBBBB - #10 Low Sodium Navy Beans'  THEN StandardCPM:=41; END_IF
IF ProductCode='5LSNOBBB - #10 Brite Low Sod Great Northern Bean'  THEN StandardCPM:=41; END_IF
IF ProductCode='5LSPBBBB - #10 Brite Low Sodium Pinto Beans'  THEN StandardCPM:=41; END_IF
IF ProductCode='5NSLKBBBB - #10 Brite Light Red Kidney Beans No Salt'  THEN StandardCPM:=41; END_IF
IF ProductCode='5PBJADKBB - #10 Brite Jalapeno Pinto Beans Dickeys'  THEN StandardCPM:=41; END_IF
IF ProductCode='5PNBBB - #10 Brite Boiled Peanuts'  THEN StandardCPM:=41; END_IF
IF ProductCode='5RBBBB - #10 Brite Red Beans'  THEN StandardCPM:=41; END_IF
IF ProductCode='5RSBBBB - #10 Brite Ranch Style Black Beans'  THEN StandardCPM:=41; END_IF
IF ProductCode='5RSPTBBB - #10 Brite Ranch Style Pinto Beans'  THEN StandardCPM:=41; END_IF
IF ProductCode='5SBEBBB - #10 Brite Seas Blackeye Peas'  THEN StandardCPM:=41; END_IF
IF ProductCode='5SFSBBB - #10 Brite Seas Field Peas/Snaps CR'  THEN StandardCPM:=41; END_IF
IF ProductCode='5SPBBBB - #10 Brite Seas Pinto Beans'  THEN StandardCPM:=41; END_IF
IF ProductCode='5GSCGBFB - #10 Brite Glory Seas FatBK Collard Green'  THEN StandardCPM:=29; END_IF
IF ProductCode='5GSMGBFB - #10 Brite Glory Seas FatBK Mixed Greens'  THEN StandardCPM:=29; END_IF
IF ProductCode='5GSTCGBB - #10 Brite Glory Seas Turkey Collard Grns'  THEN StandardCPM:=29; END_IF
IF ProductCode='5NCGBBB - #10 Brite Collard Greens NSA'  THEN StandardCPM:=29; END_IF
IF ProductCode='5NKABBB - #10 Brite No Salt Kale Greens'  THEN StandardCPM:=29; END_IF
IF ProductCode='5NMGBBB - #10 Brite Mixed Greens NSA'  THEN StandardCPM:=29; END_IF
IF ProductCode='5NMUDMBBB - #10 Brite Allens Mustard Greens NSA'  THEN StandardCPM:=29; END_IF
IF ProductCode='5NTGBBB - #10 Brite Turnip Greens NSA'  THEN StandardCPM:=29; END_IF
IF ProductCode='5SCGBBB - #10 Brite Seas Collard Greens'  THEN StandardCPM:=29; END_IF
IF ProductCode='5SMIGBBB - #10 Brite Seas Mixed Greens'  THEN StandardCPM:=29; END_IF
IF ProductCode='5STGBBB - #10 Brite Seas Turnip Greens'  THEN StandardCPM:=29; END_IF
IF ProductCode='5PNBDMBBB - #10 Brite Pork and Beans'  THEN StandardCPM:=33; END_IF
IF ProductCode='5VCPBBB - #10 Brite Van Camps Pork & Beans'  THEN StandardCPM:=33; END_IF
IF ProductCode='5VEGBKBDMBB - #10 Brite Allens Vegetarian Baked Beans'  THEN StandardCPM:=33; END_IF
IF ProductCode='5VEGBNBBB - #10 Brite Allens Vegetarian Beans'  THEN StandardCPM:=33; END_IF
IF ProductCode='5MEXCHBNBB - #10 Brite Mexican Chili Beans'  THEN StandardCPM:=33; END_IF
IF ProductCode='5ALLSNSVEGBBB - #10 Brite Allens LS NS Veg Beans'  THEN StandardCPM:=33; END_IF
IF ProductCode='5BBNHBBB - #10 Brite Hattie Bs Baked Beans'  THEN StandardCPM:=33; END_IF
IF ProductCode='5BKBNBBB - #10 Brite DM Baked Beans'  THEN StandardCPM:=33; END_IF
IF ProductCode='5BKBNSCBBB - #10 Brite Slow Cooked Baked Beans'  THEN StandardCPM:=33; END_IF
IF ProductCode='5BQBNDKBB - #10 Brite BarB Q Beans Dickeys'  THEN StandardCPM:=33; END_IF
IF ProductCode='5HCPNBBB - #10 Brite Happy Chef Pork and Beans'  THEN StandardCPM:=33; END_IF
IF ProductCode='5SQCBBB - #10 Brite Yellow Squash 1" Cut'  THEN StandardCPM:=27; END_IF
IF ProductCode='5SQOBBB - #10 Brite Yellow Squash Cut w/Onions'  THEN StandardCPM:=27; END_IF
IF ProductCode='5LSSIBBB - #10 Brite Spinach Chopped 1/2" x 1/2"'  THEN StandardCPM:=24; END_IF
IF ProductCode='5NSIBBB - #10 Brite Spinach NSA Cut Leaf  ¾" x ¾"'  THEN StandardCPM:=24; END_IF
IF ProductCode='5NTWBBB - #10 Brite Turnips with Roots NSA'  THEN StandardCPM:=24; END_IF
IF ProductCode='5SCBBB - #10 Brite Spinach Leaf 3/4" x 3/4"'  THEN StandardCPM:=24; END_IF
IF ProductCode='5PDIBBB - #10 Brite White Diced Potatoes'  THEN StandardCPM:=36; END_IF
IF ProductCode='5RUTBBB - #10 Brite Diced Rutabagas'  THEN StandardCPM:=36; END_IF
IF ProductCode='5ITBBBB - #10 Brite Italian Green Beans'  THEN StandardCPM:=30; END_IF
IF ProductCode='5ITSENBBB - #10 Brite MH Italian Grn Beans USF'  THEN StandardCPM:=30; END_IF
IF ProductCode='5YCANDBB - #10 Brite Candied Yams'  THEN StandardCPM:=30; END_IF
IF ProductCode='5YCT4555BB - #10 Brite Cut Yams 45/55 Count'  THEN StandardCPM:=30; END_IF
IF ProductCode='5YCTELBBB - #10 Extra Light Syrup Cut Yams'  THEN StandardCPM:=30; END_IF
IF ProductCode='5SITBDKBB - #10 Brite Sea Italian Grn Beans Dickeys'  THEN StandardCPM:=30; END_IF
IF ProductCode='5SITBBBB - #10 Brite Seasoned Italian Green Beans'  THEN StandardCPM:=30; END_IF
IF ProductCode='5ALSBNBBB - #10 Brite Allens Seas Cut Green Beans'  THEN StandardCPM:=30; END_IF
IF ProductCode='5ALSITBBB - #10 Brite Allens Seas Ital Green Beans'  THEN StandardCPM:=30; END_IF
IF ProductCode='5BNBBB - #10 Brite Green Beans Cut'  THEN StandardCPM:=30; END_IF
IF ProductCode='5BNCBBBB - #10 Brite Cracker Barrel Green Beans Cut'  THEN StandardCPM:=30; END_IF
IF ProductCode='5SBNBBB - #10 Brite Seasoned Cut Green Beans'  THEN StandardCPM:=30; END_IF
IF ProductCode='5VAMVBBB - #10 Brite Veg-All Mixed Vegetables'  THEN StandardCPM:=38; END_IF
IF ProductCode='5YMASBBB - #10 Brite Mashed Yams'  THEN StandardCPM:=14; END_IF

END_FUNCTION_BLOCK

// ---- POUs/Status_and_Alarms.TcPOU
PROGRAM Status_and_Alarms
VAR

END_VAR

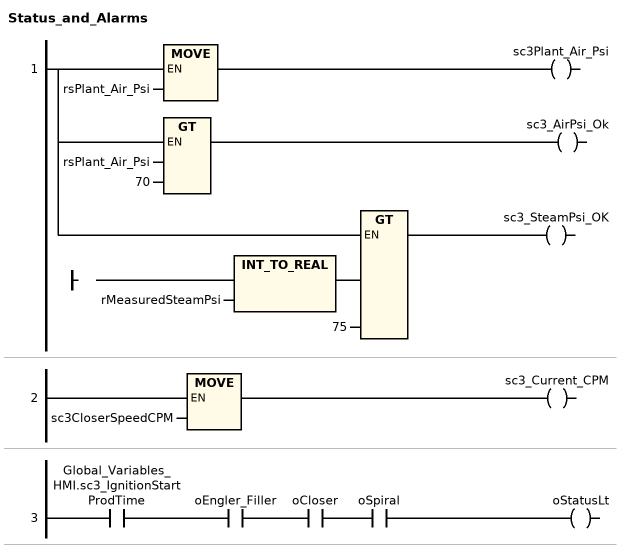
// NETWORK 1
sc3Plant_Air_Psi := rsPlant_Air_Psi;
sc3_AirPsi_Ok := rsPlant_Air_Psi > 70;
sc3_SteamPsi_OK := INT_TO_REAL(rMeasuredSteamPsi) > 75;

// NETWORK 2
sc3_Current_CPM := sc3CloserSpeedCPM;

// NETWORK 3
oStatusLt := Global_Variables_HMI.sc3_IgnitionStartProdTime AND oEngler_Filler AND oCloser AND oSpiral;

END_PROGRAM

// ---- POUs/Runtime_Control.TcPOU
PROGRAM Runtime_Control
VAR
	RuntimeActivate: BOOL;
	FRA3RT: Production_Runtime_Values;
	BackupCanCounterA: CTU;
	BackCanCounterA_CurrentCount: WORD;
	ResetBackupCounterA: BOOL;
	BackupCanCounterB: CTU;
	BackCanCounterB_CurrentCount: WORD;
	MultiplierValue_FOR_BackupCounterB: DINT;

	FRA3_Downtime_LOG: FB_Downtime_LOG;
	DowntimeDetected: BOOL;
	ResetStopReasonsValues: F_TRIG;
END_VAR

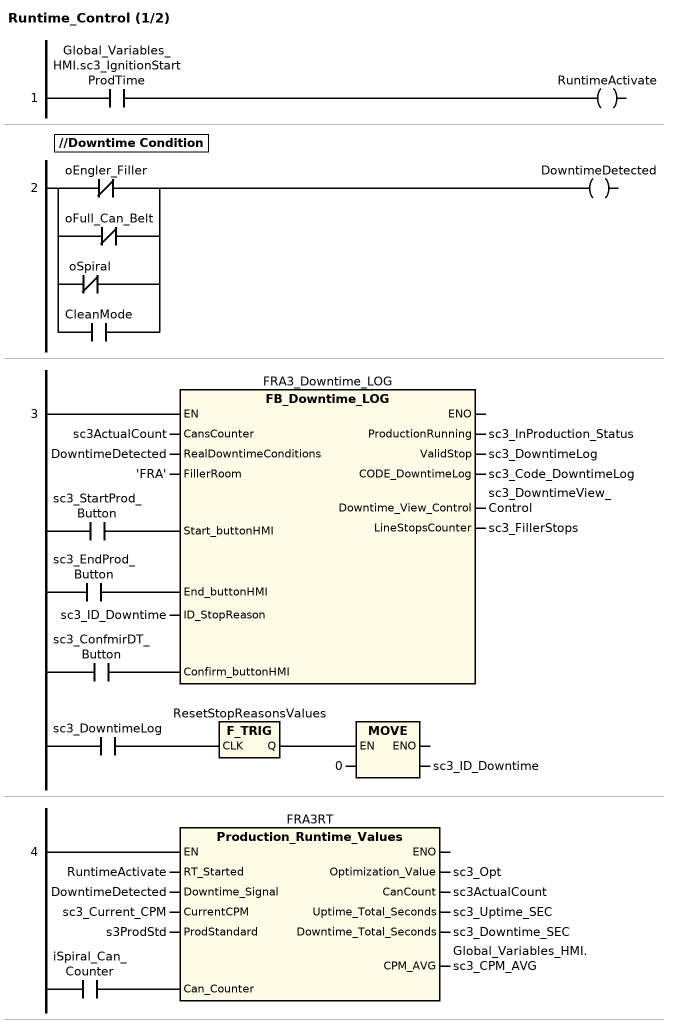
// NETWORK 1
RuntimeActivate := Global_Variables_HMI.sc3_IgnitionStartProdTime;

// NETWORK 2
// label: //Downtime Condition
DowntimeDetected := NOT oEngler_Filler OR NOT oFull_Can_Belt OR NOT oSpiral OR CleanMode;

// NETWORK 3
FRA3_Downtime_LOG(
    CansCounter := sc3ActualCount,
    RealDowntimeConditions := DowntimeDetected,
    FillerRoom := 'FRA',
    Start_buttonHMI := sc3_StartProd_Button,
    End_buttonHMI := sc3_EndProd_Button,
    ID_StopReason := sc3_ID_Downtime,
    Confirm_buttonHMI := sc3_ConfmirDT_Button,
    ProductionRunning => sc3_InProduction_Status,
    ValidStop => sc3_DowntimeLog,
    CODE_DowntimeLog => sc3_Code_DowntimeLog,
    Downtime_View_Control => sc3_DowntimeView_Control,
    LineStopsCounter => sc3_FillerStops); // FB_Downtime_LOG
ResetStopReasonsValues(CLK := sc3_DowntimeLog); // F_TRIG
IF ResetStopReasonsValues.Q THEN sc3_ID_Downtime := 0; END_IF

// NETWORK 4
FRA3RT(
    RT_Started := RuntimeActivate,
    Downtime_Signal := DowntimeDetected,
    CurrentCPM := sc3_Current_CPM,
    ProdStandard := s3ProdStd,
    Can_Counter := iSpiral_Can_Counter,
    Optimization_Value => sc3_Opt,
    CanCount => sc3ActualCount,
    Uptime_Total_Seconds => sc3_Uptime_SEC,
    Downtime_Total_Seconds => sc3_Downtime_SEC,
    CPM_AVG => Global_Variables_HMI.sc3_CPM_AVG); // Production_Runtime_Values

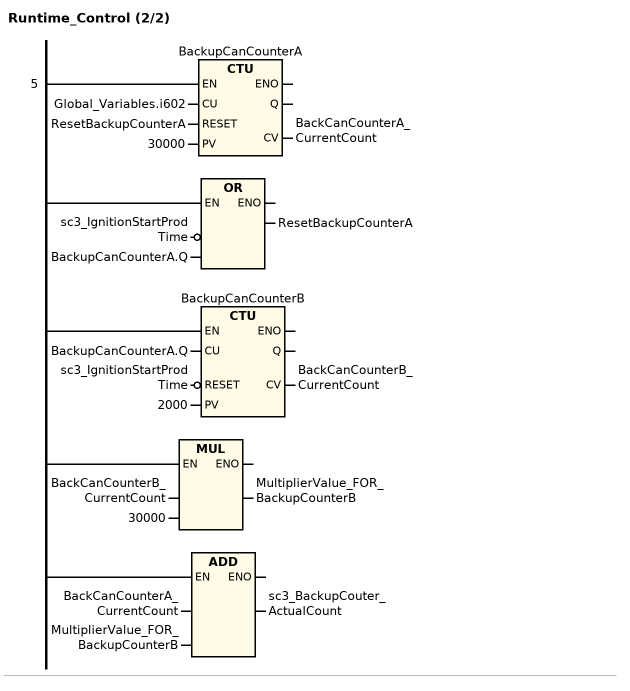
// NETWORK 5
BackupCanCounterA(
    CU := Global_Variables.i602,
    RESET := ResetBackupCounterA,
    PV := 30000,
    CV => BackCanCounterA_CurrentCount); // CTU
ResetBackupCounterA := NOT sc3_IgnitionStartProdTime OR BackupCanCounterA.Q;
BackupCanCounterB(
    CU := BackupCanCounterA.Q,
    RESET := NOT sc3_IgnitionStartProdTime,
    PV := 2000,
    CV => BackCanCounterB_CurrentCount); // CTU
MultiplierValue_FOR_BackupCounterB := BackCanCounterB_CurrentCount * 30000;
sc3_BackupCouter_ActualCount := BackCanCounterA_CurrentCount + MultiplierValue_FOR_BackupCounterB;

END_PROGRAM

// ---- POUs/Production_Runtime_Values.TcPOU
FUNCTION_BLOCK Production_Runtime_Values
VAR_INPUT
	RT_Started:BOOL;
	Downtime_Signal:BOOL;
	CurrentCPM:REAL;
	ProdStandard:REAL;
	Can_Counter:BOOL;
	
END_VAR
VAR_OUTPUT

	Optimization_Value:REAL;
	CanCount:REAL;
	Uptime_Total_Seconds: DINT;
	Downtime_Total_Seconds: DINT;
	CPM_AVG: REAL;
END_VAR
VAR
	CanCounter: CTU;
	CanCounterMultiplier: CTU;
	CanMultiplierCount: WORD;

	CanCountCurrent: WORD;
	CurrentCanCount: INT;
	Multiplier_CanCountV: REAL;
	CanCountValueB: INT;
	sc_TotalCanCount: INT;
	RT1: tof;
	RT2: TOF;
	Runtime_Value: CTU;
	Spent_Production_Time: WORD;
	SpentProductionTime: INT;

	AdjustedCPM: INT;
	CansEstimatedToBeRun: REAL;
	Opt_ValueA: REAL;
	Opt_before_10: REAL;
	OPTA: INT;
	CheckDivA: CheckDiv_1;
	Estimated_Cans: REAL;
	OptValue_A: REAL;
	Reset: BOOL;
	VerifyDivider: CheckDiv_1;
	SPTReal: REAL;
	
	Downtime_TimeAccumulator: GetTime_Seconds;
	Uptime_TimeAccumulator: GetTime_Seconds;
END_VAR

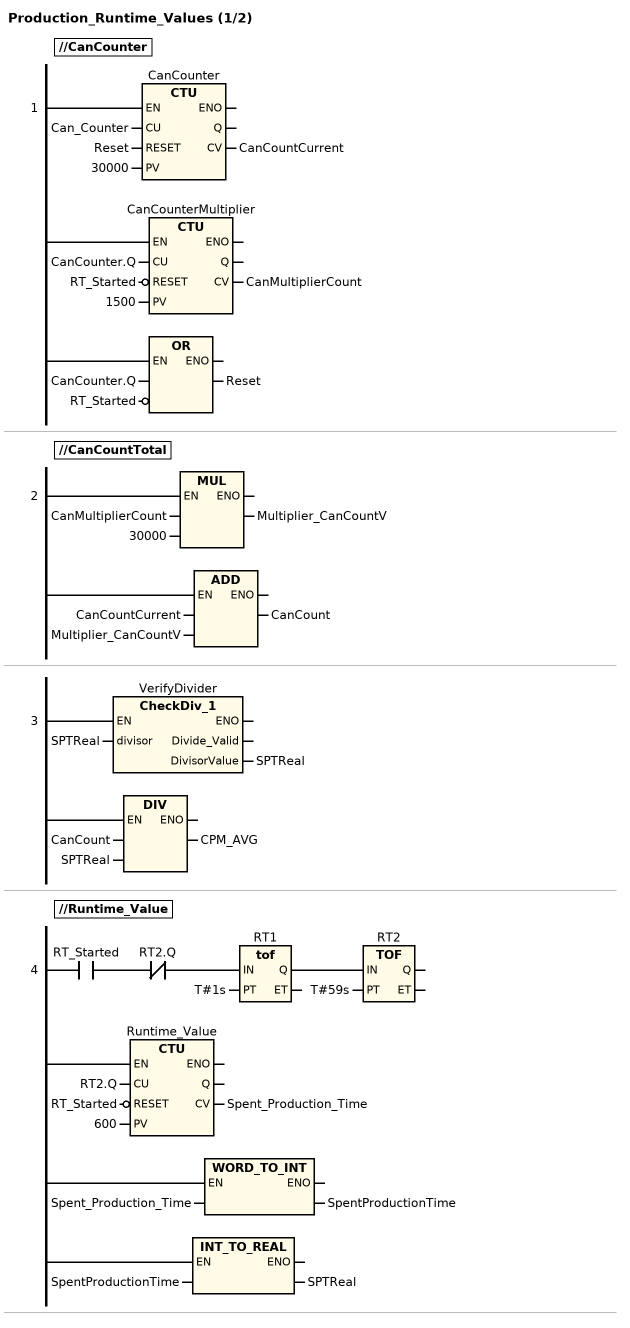
// NETWORK 1
// label: //CanCounter
CanCounter(CU := Can_Counter, RESET := Reset, PV := 30000, CV => CanCountCurrent); // CTU
CanCounterMultiplier(CU := CanCounter.Q, RESET := NOT RT_Started, PV := 1500, CV => CanMultiplierCount); // CTU
Reset := CanCounter.Q OR NOT RT_Started;

// NETWORK 2
// label: //CanCountTotal
Multiplier_CanCountV := CanMultiplierCount * 30000;
CanCount := CanCountCurrent + Multiplier_CanCountV;

// NETWORK 3
VerifyDivider(divisor := SPTReal, DivisorValue => SPTReal); // CheckDiv_1
CPM_AVG := CanCount / SPTReal;

// NETWORK 4
// label: //Runtime_Value
RT1(IN := RT_Started AND NOT RT2.Q, PT := T#1s); // tof
RT2(IN := RT1.Q, PT := T#59s); // TOF
Runtime_Value(CU := RT2.Q, RESET := NOT RT_Started, PV := 600, CV => Spent_Production_Time); // CTU
SpentProductionTime := WORD_TO_INT(Spent_Production_Time);
SPTReal := INT_TO_REAL(SpentProductionTime);

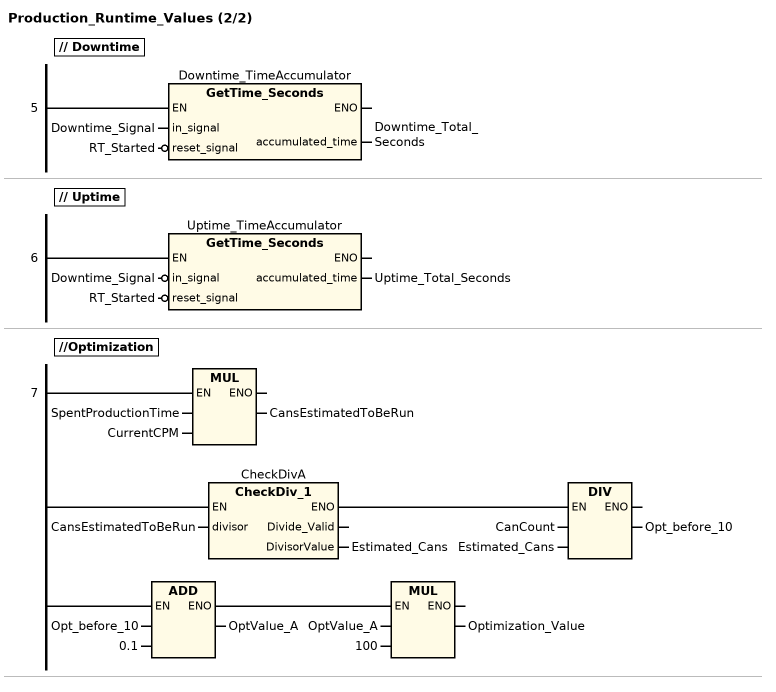
// NETWORK 5
// label: // Downtime
Downtime_TimeAccumulator(
    EN := TRUE,
    in_signal := Downtime_Signal,
    reset_signal := NOT RT_Started,
    accumulated_time => Downtime_Total_Seconds); // GetTime_Seconds

// NETWORK 6
// label: // Uptime
Uptime_TimeAccumulator(
    EN := TRUE,
    in_signal := NOT Downtime_Signal,
    reset_signal := NOT RT_Started,
    accumulated_time => Uptime_Total_Seconds); // GetTime_Seconds

// NETWORK 7
// label: //Optimization
CansEstimatedToBeRun := SpentProductionTime * CurrentCPM;
CheckDivA(divisor := CansEstimatedToBeRun, DivisorValue => Estimated_Cans); // CheckDiv_1
Opt_before_10 := CanCount / Estimated_Cans;
OptValue_A := Opt_before_10 + 0.1;
Optimization_Value := OptValue_A * 100;

END_FUNCTION_BLOCK

// ---- POUs/Function Blocks/CheckDiv_1.TcPOU
FUNCTION_BLOCK CheckDiv_1
VAR_INPUT
    divisor : REAL;
END_VAR
VAR_OUTPUT
	Divide_Valid:BOOL;
	DivisorValue:REAL;
	
END_VAR
VAR
	CheckDivReal: REAL;
END_VAR

IF divisor = 0 THEN
    DivisorValue := 1;
	
ELSE
	DivisorValue := divisor;
END_IF

END_FUNCTION_BLOCK

// ---- POUs/Function Blocks/GetTime_Seconds.TcPOU
FUNCTION_BLOCK GetTime_Seconds
VAR_INPUT
	EN: BOOL;
	in_signal: BOOL;
	reset_signal: BOOL;
END_VAR
VAR_OUTPUT
	ENO: BOOL;
	accumulated_time: DINT;
END_VAR
VAR	
	cycle_count: DINT;
END_VAR

ENO:=EN;
IF NOT EN THEN
	RETURN;
END_IF

IF reset_signal THEN
	cycle_count := 0;
	accumulated_time:=0;
END_IF

IF in_signal THEN
	cycle_count := cycle_count + 1; 
END_IF

accumulated_time:= cycle_count / 100; // cycle task=10m

END_FUNCTION_BLOCK

// ---- POUs/Function Blocks/FB_Downtime_LOG.TcPOU
FUNCTION_BLOCK FB_Downtime_LOG
VAR_INPUT
	CansCounter: REAL;
	RealDowntimeConditions: BOOL;
	FillerRoom: STRING;
	Start_buttonHMI: BOOL;
	End_buttonHMI: BOOL;
	ID_StopReason: INT; 
	Confirm_buttonHMI: BOOL;
	
END_VAR
VAR_OUTPUT
	ProductionRunning: BOOL;
	ValidStop: BOOL; //DowntimeLog: BOOL;
	CODE_DowntimeLog: STRING;
	Downtime_View_Control: BOOL;
	LineStopsCounter: INT;
	
	
END_VAR
VAR
	FixedSchedule_Verify: FixedSchedule_FillerRoom;
	onSchedule: BOOL;
	StartButton: R_TRIG;
	RedCan_Button: R_TRIG;
	
	StartedCounter: BOOL;
	RS_Dowtime: RS;
	Reset_DowntimeLog: BOOL;
	DT_Confirm_Button: R_TRIG;
	DT_ConfirmB: BOOL;
	
 	RealStop: BOOL;
	
	ValidStop_Verifier: TON;
	PulseHMI_StopScreen: TP;
	Codes_StopReason_HMI: Codes_StopReason;
	VALID_StopCode: BOOL;
	SaveStopReasonsValues: R_TRIG;
	StopNumber: INT;	
	FillerStopped: CTU; //Counter stops
	CansDetected: R_TRIG;
END_VAR

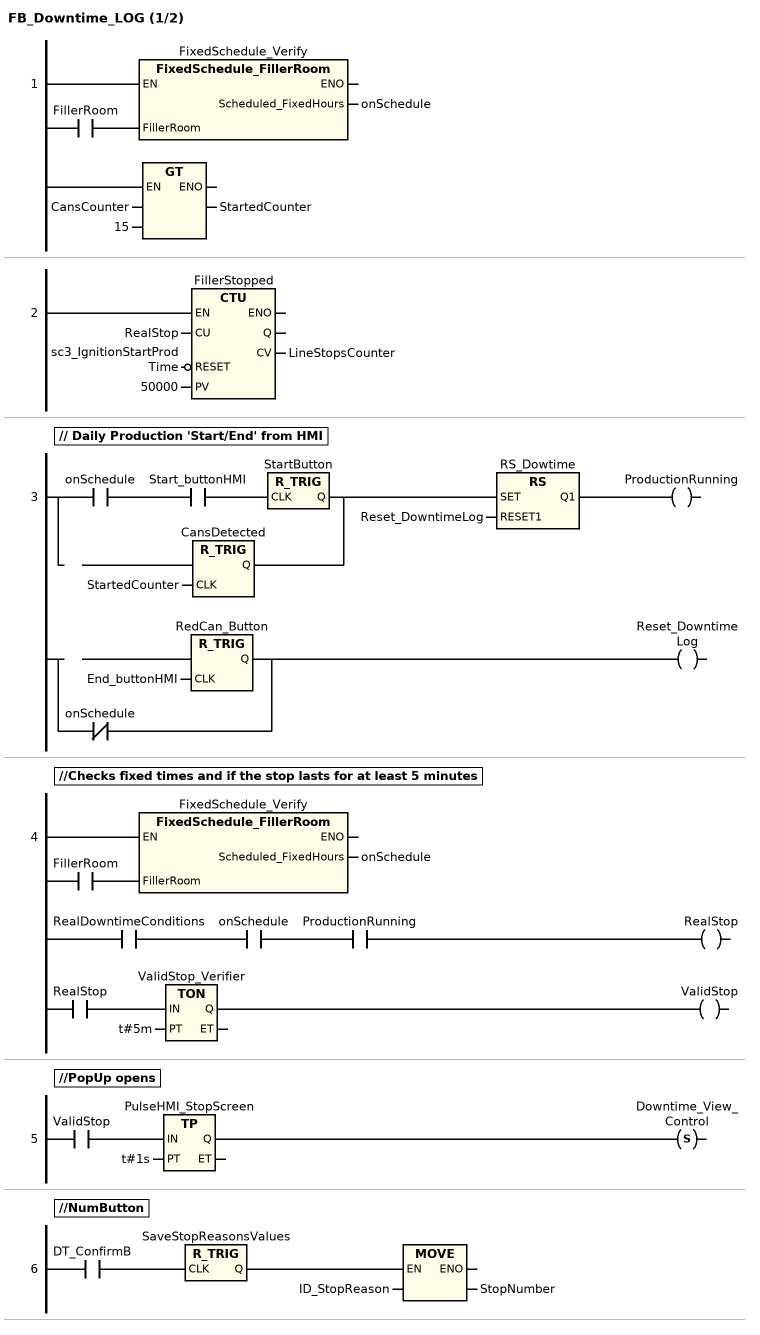
// NETWORK 1
FixedSchedule_Verify(FillerRoom := FillerRoom, Scheduled_FixedHours => onSchedule); // FixedSchedule_FillerRoom
StartedCounter := CansCounter > 15;

// NETWORK 2
FillerStopped(CU := RealStop, RESET := NOT sc3_IgnitionStartProdTime, PV := 50000, CV => LineStopsCounter); // CTU

// NETWORK 3
// label: // Daily Production 'Start/End' from HMI
StartButton(CLK := onSchedule AND Start_buttonHMI); // R_TRIG
CansDetected(CLK := StartedCounter); // R_TRIG
RS_Dowtime(SET := StartButton.Q OR CansDetected.Q, RESET1 := Reset_DowntimeLog); // RS
ProductionRunning := RS_Dowtime.Q1;
RedCan_Button(CLK := End_buttonHMI); // R_TRIG
Reset_DowntimeLog := RedCan_Button.Q OR NOT onSchedule;

// NETWORK 4
// label: //Checks fixed times and if the stop lasts for at least 5 minutes
FixedSchedule_Verify(FillerRoom := FillerRoom, Scheduled_FixedHours => onSchedule); // FixedSchedule_FillerRoom
RealStop := (RealDowntimeConditions AND onSchedule) AND ProductionRunning;
ValidStop_Verifier(IN := RealStop, PT := t#5m); // TON
ValidStop := ValidStop_Verifier.Q;

// NETWORK 5
// label: //PopUp opens
PulseHMI_StopScreen(IN := ValidStop, PT := t#1s); // TP
Downtime_View_Control S= PulseHMI_StopScreen.Q;

// NETWORK 6
// label: //NumButton
SaveStopReasonsValues(CLK := DT_ConfirmB); // R_TRIG
IF SaveStopReasonsValues.Q THEN StopNumber := ID_StopReason; END_IF

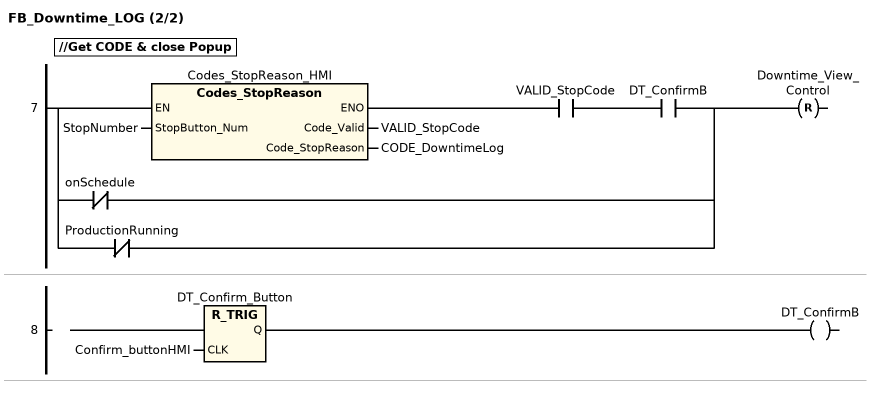
// NETWORK 7
// label: //Get CODE & close Popup
Codes_StopReason_HMI(
    EN := TRUE,
    StopButton_Num := StopNumber,
    Code_Valid => VALID_StopCode,
    Code_StopReason => CODE_DowntimeLog); // Codes_StopReason
Downtime_View_Control R= TRUE AND VALID_StopCode AND DT_ConfirmB OR NOT onSchedule OR NOT ProductionRunning;

// NETWORK 8
DT_Confirm_Button(CLK := Confirm_buttonHMI); // R_TRIG
DT_ConfirmB := DT_Confirm_Button.Q;

END_FUNCTION_BLOCK

// ---- POUs/Function Blocks/FixedSchedule_FillerRoom.TcPOU
FUNCTION_BLOCK FixedSchedule_FillerRoom
VAR_INPUT
	FillerRoom: STRING;
END_VAR

VAR_OUTPUT
	Scheduled_FixedHours: BOOL;
END_VAR
	
VAR
	total_minutes: INT;
	fbTime : FB_LocalSystemTime;
    stTime : TIMESTRUCT;
	Current_Hours: WORD; 
	Current_Minutes: WORD;
	
END_VAR

//Current time
fbTime(
    sNetID := '',
    bEnable := TRUE,
    dwCycle := 1000
);

stTime := fbTime.systemTime;
Current_Hours :=  stTime.wHour;
Current_Minutes := stTime.wMinute;


total_minutes := (WORD_TO_INT(Current_Hours) * 60) +
                  WORD_TO_INT(Current_Minutes);

// Shift per Filler Room
IF FillerRoom = 'FRA' OR FillerRoom = 'FRD'THEN
	Scheduled_FixedHours:= NOT((total_minutes>=120)AND(total_minutes<360)); //02:00am to 05:59 //(add 20 min after 2:00am just in case)
ELSIF  FillerRoom = 'FRC' THEN
	Scheduled_FixedHours:= NOT((total_minutes>=150)AND(total_minutes<390)); //02:30am to 06:29 //(add 20 min after 2:30am just in case)
ELSE
	Scheduled_FixedHours:= FALSE;
END_IF;

END_FUNCTION_BLOCK

// ---- POUs/Function Blocks/Codes_StopReason.TcPOU
FUNCTION_BLOCK Codes_StopReason
VAR_INPUT
	EN: BOOL;
	StopButton_Num : INT;       
END_VAR
VAR_OUTPUT
	ENO: BOOL;
	Code_Valid: BOOL;
	Code_StopReason : STRING;  
	
	
END_VAR
VAR
	
END_VAR

IF NOT EN THEN
    ENO := FALSE;
    Code_StopReason := '';
    Code_Valid := FALSE;
    RETURN;
END_IF

ENO := TRUE;

CASE StopButton_Num OF
    10: Code_StopReason := 'MNT_C01';
    20: Code_StopReason := 'MNT_G01';
    30: Code_StopReason := 'MSP_C01';
    40: Code_StopReason := 'MSP_P01';
    50: Code_StopReason := 'QLT_Q01';
    60: Code_StopReason := 'TEC_E0M';
	70: Code_StopReason := 'MSP_F01';
ELSE
    Code_StopReason := '';
END_CASE;

Code_Valid := (Code_StopReason <> '');

END_FUNCTION_BLOCK

// ---- POUs/Function Blocks/CounterEx.TcPOU
FUNCTION_BLOCK CounterEx
VAR_INPUT

                 CU : BOOL;

                PV: INT;

                ForcedCV : INT;

                RESET : BOOL;
					
				

END_VAR
VAR_OUTPUT

                Q : BOOL;

                CV : INT;

END_VAR
VAR

                RisingEdge : BOOL;

                LastForcedCV : INT;

END_VAR

IF (CU) AND (NOT RisingEdge) THEN

                IF (CV<2147483646) THEN

                                CV:=CV+1;

                END_IF

END_IF

RisingEdge:=CU;

 

IF (LastForcedCV<>ForcedCV) THEN

                CV:=ForcedCV;

                LastForcedCV:=ForcedCV;

END_IF

 

IF (RESET) THEN

                CV:=0;

END_IF

 

Q:=(CV>=PV);

END_FUNCTION_BLOCK
